Universal Robots PolyScope program: 958_16_OCT_2021_DER.urp

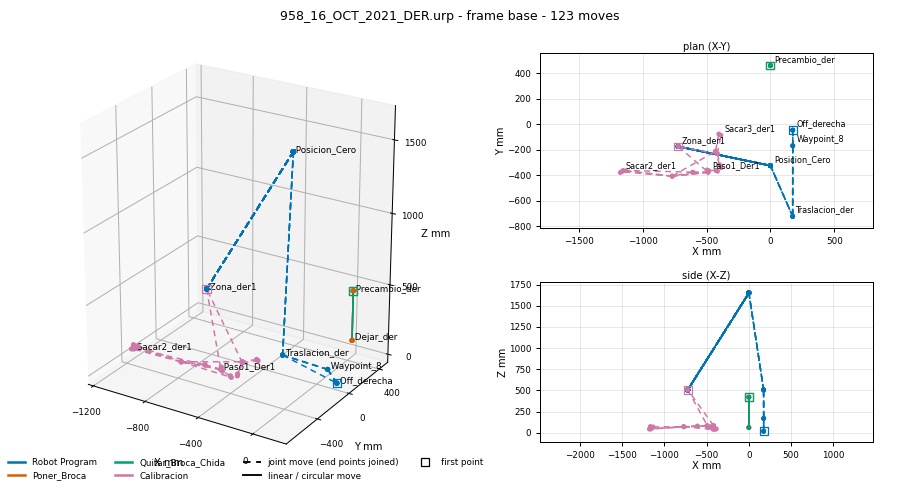
[picture p0: tool path of 958_16_OCT_2021_DER.urp in frame base, 123 of 219 moves have a stored position in this frame; points joined in program order, loops and branches not executed]
Program 958_16_OCT_2021_DER (installation=instalacion_derecha_10_MAR_21 directory=/programs/FAI3 createdIn=5.6.0.90886 lastSavedIn=5.11.1.108318 robotSerialNumber=20195001785)
Calibrated DH parameters: a=[0.000107, -0.568984, -0.552934, -0.00001, -0.000063, 0]; d=[0.180718, -257.998067, 200.685024, 57.48776, 0.119923, 0.115353]; alpha=[1.571119, 0.000876, -0.002498, 1.571178, -1.570523, 0]; deltaTheta=[0, -0.378191, 0.631587, -0.253396, 0, 0]
Robot Program (runOnlyOnce=false)
  SuppressedNode
    Folder Pruebas_Cambiador
      MoveJ speed 30 deg/s, acceleration 50 deg/s^2 (useActiveTCP=true) feature=Base
        Waypoint Precambio_der: TCP in base x=0.184 y=459.545 z=420.003 mm, rx=0.2788 ry=3.1256 rz=-0.0305 rad; joints [126.473, -59.389, -120.459, -180.773, -48.503, 0.207] deg; TCP offset x=0.151 y=-167.165 z=35.088 mm, rx=1.5784 ry=-0.0729 rz=0.0687 rad
      Loop Forever
        Call Poner_Broca
        Call Quitar_Broca_Chida
  SuppressedNode
    'Codigo'
  Set DigitalOutput pin=digital_out[0]; digitalValue=1
  MoveJ speed 30 deg/s, acceleration 50 deg/s^2 (useActiveTCP=true) feature=Base
    Waypoint Off_derecha: TCP in base x=175.178 y=-46.666 z=17.814 mm, rx=-1.9982 ry=0.0913 rz=0.0579 rad; joints [90, -90, 154.891, 0, 90, 0.001] deg
  broca := 1645
  Script: textmsg("----------DAS-----------")
  If Lado_Correr≟2
    If pos_sig_der≟0
      Folder Arranque
        Set ExpressionOutput pin=mensaje_mw10; expression=15
        Wait DigitalInput pin=Continuar_M30; digitalValue=1
        Wait Sleep waitTime=1
        MoveJ speed 60 deg/s, acceleration 80 deg/s^2 (useActiveTCP=true) feature=Base
          Waypoint Off_derecha: TCP in base x=175.178 y=-46.666 z=17.814 mm, rx=-1.9982 ry=0.0913 rz=0.0579 rad; joints [90, -90, 154.891, 0, 90, 0.001] deg
        Set DigitalOutput pin=postrnas_m187; digitalValue=1
        Wait Sleep waitTime=1
        Set DigitalOutput pin=Home_M20; digitalValue=1
        Wait Sleep waitTime=1
        Set DigitalOutput pin=postrnas_m187; digitalValue=0
        Set DigitalOutput pin=Home_M20; digitalValue=0
        Set ExpressionOutput pin=mensaje_mw10; expression=20
        Wait DigitalInput pin=Continuar_M30; digitalValue=1
        Wait Sleep waitTime=1
      Folder Traslacion
        Set ExpressionOutput pin=mensaje_mw10; expression=25
        Wait DigitalInput pin=Continuar_M30; digitalValue=1
        Wait Sleep waitTime=1
        MoveJ speed 60 deg/s, acceleration 80 deg/s^2 (useActiveTCP=true) feature=Base
          Waypoint Waypoint_8: TCP in base x=175.237 y=-168.919 z=168.903 mm, rx=3.0585 ry=-0.1387 rz=0.0062 rad; joints [90.001, -160.001, 154.893, -0.003, 90, 0.003] deg
          Waypoint Traslacion_der: TCP in base x=174.612 y=-721.747 z=506.267 mm, rx=3.1383 ry=-0.1432 rz=0.0001 rad; joints [89.991, -90.247, 90.386, -0.667, 89.974, 0.014] deg
        Set ExpressionOutput pin=mensaje_mw10; expression=30
        Wait DigitalInput pin=Continuar_M30; digitalValue=1
        Wait Sleep waitTime=1
        Set DigitalOutput pin=postrnas_m187; digitalValue=1
        Wait Sleep waitTime=1
        Set DigitalOutput pin=pose2_m252; digitalValue=1
        Wait Sleep waitTime=1
        Set DigitalOutput pin=pose2_m252; digitalValue=0
        Set DigitalOutput pin=postrnas_m187; digitalValue=0
        Wait Sleep waitTime=10
        Set ExpressionOutput pin=mensaje_mw10; expression=35
        Wait DigitalInput pin=Continuar_M30; digitalValue=1
        Wait Sleep waitTime=1
      Folder Brocas
        Set DigitalOutput pin=carrusel_home; digitalValue=1
        Wait Sleep waitTime=1
        Set DigitalOutput pin=carrusel_home; digitalValue=0
        Set ExpressionOutput pin=mensaje_mw10; expression=40
        Wait DigitalInput pin=Continuar_M30; digitalValue=1
        Wait Sleep waitTime=1
        Set DigitalOutput pin=carrusel_home; digitalValue=1
        Wait Sleep waitTime=1
        Set DigitalOutput pin=carrusel_home; digitalValue=0
        Set ExpressionOutput pin=mensaje_mw10; expression=45
        Wait DigitalInput pin=Continuar_M30; digitalValue=1
        Wait Sleep waitTime=1
        Call Poner_Broca
      Folder Offsets factor
        SuppressedNode
          broca := 1645
        L1B1x := ((0.09525254)/(0.09525))*(0.09525254)
        L1B1y := ((-0.01266698)/(-0.0127))*(-0.01266698)
        L1B2x := ((0.75576176)/(0.75565))*(0.75576176)
        L1B2y := ((-0.01269238)/(-0.0127))*(-0.01269238)
        L2B1x := ((0.09513062)/(0.09525))*(0.09525)
        L2B1y := ((0.39369238)/(0.3937))*(0.39369238)
        L2B2x := ((0.75565508)/(0.75565))*(0.75565508)
        L2B2y := ((0.39372032)/(0.3937))*(0.39372032)
      Folder Calibracion
        Set ExpressionOutput pin=mensaje_mw10; expression=50
        Wait DigitalInput pin=Continuar_M30; digitalValue=1
        Wait Sleep waitTime=1
        MoveJ speed 60 deg/s, acceleration 80 deg/s^2 (useActiveTCP=true) feature=Base
          Waypoint Posicion_Cero: TCP in base x=0.641 y=-324.742 z=1651.532 mm, rx=-0.0042 ry=-0.0154 rz=-3.0499 rad; joints [-0.001, -90.003, -0.001, -90, 0, 0.002] deg
          Waypoint Zona_der1: TCP in base x=-721.714 y=-174.597 z=506.289 mm, rx=2.1128 ry=-2.325 rz=0 rad; joints [0.057, -90.231, 90.368, -0.664, 90.292, 0.009] deg
        broca := 1645
        Set ExpressionOutput pin=mensaje_mw10; expression=125
        Wait DigitalInput pin=Continuar_M30; digitalValue=1
        Wait Sleep waitTime=1
        Set ExpressionOutput pin=mensaje_mw10; expression=130
        Wait DigitalInput pin=Continuar_M30; digitalValue=1
        Wait Sleep waitTime=1
        Call Calibracion
      Folder GoNoGo
        Set ExpressionOutput pin=mensaje_mw10; expression=55
        Wait DigitalInput pin=Continuar_M30; digitalValue=1
        Wait Sleep waitTime=1
        Set ExpressionOutput pin=mensaje_mw10; expression=60
        Wait DigitalInput pin=Continuar_M30; digitalValue=1
        Wait Sleep waitTime=1
        Folder Linea1_Buje1
          Xfin := (((L1B1x)*Xp)-(Xd)-((L1B1y)*(1/m2)))*(-1)
          Yfin := (((L1B1y)*Yp)-(Yd)+((L1B1x)*m1))*(-1)
          rotaciones := get_actual_tcp_pose()
          var_3 := rotaciones[3]
          var_4 := rotaciones[4]
          var_5 := rotaciones[5]
          If broca≟1645
            PosFinal := p[Xfin+0.00208915,Yfin+0.00208915,0.1,var_3,var_4,var_5]
          ElseIf broca≟1935
            PosFinal := p[Xfin+0.00245745,Yfin+0.00245745,0.1,var_3,var_4,var_5]
          ElseIf broca≟217
            PosFinal := p[Xfin+0.0027559,Yfin+0.0027559,0.1,var_3,var_4,var_5]
          Buje_Final := PosFinal
        MoveJ speed 60 deg/s, acceleration 80 deg/s^2 (useActiveTCP=true) feature=Base
          Waypoint Waypoint (Variable): variable(name=Buje_Final)
        Wait Sleep waitTime=1
        Folder Alturas
          If P1h[2]<P2h[2]
            tcp := get_actual_tcp_pose()
            offset_altura := p[tcp[0],tcp[1],((alta-0.0095)-(altura/1000)),tcp[3],tcp[4],tcp[5]]
            MoveL speed 250 mm/s, acceleration 1200 mm/s^2 (useActiveTCP=true) feature=Base
              Waypoint Waypoint (Variable): motionParameters(jointSpeed=1.047198 jointAcceleration=1.396263 cartesianSpeed=0.03 cartesianAcceleration=0.04); variable=offset_altura
          Else 
            tcp := get_actual_tcp_pose()
            offset_altura := p[tcp[0],tcp[1],((alta-0.0095)),tcp[3],tcp[4],tcp[5]]
            MoveL speed 250 mm/s, acceleration 1200 mm/s^2 (useActiveTCP=true) feature=Base
              Waypoint Waypoint (Variable): motionParameters(jointSpeed=1.047198 jointAcceleration=1.396263 cartesianSpeed=0.03 cartesianAcceleration=0.04); variable=offset_altura
        MoveL speed 60 mm/s, acceleration 80 mm/s^2 (useActiveTCP=true) feature=Base
          Folder Freemove
            Wait Sleep waitTime=2
            Script: freedrive_mode()
            Wait Sleep waitTime=2.5
            Script: end_freedrive_mode()
            var_11 := get_actual_tcp_pose()
            var_11 := p[var_11[0]*1000,var_11[1]*1000,420,420,420,420]
            var_11 := get_actual_tcp_pose()
            var_11 := p[var_11[0],var_11[1],0.1,var_11[3],var_11[4],var_11[5]]
          MoveDirectionNode (selectedDirection=ZPlus)
            Until DISTANCE (allowActions=false deceleration=3 distanceNodeType=STOP) Distance=0.15; motionParameters(blendRadius=0)
          MoveDirectionNode (selectedDirection=XMinus)
            Until DISTANCE (allowActions=false deceleration=3 distanceNodeType=STOP) Distance=0.42; motionParameters(blendRadius=0)
        L1B1 := var_11
        Folder Linea1_Buje2
          Xfin := (((L1B2x)*Xp)-(Xd)-((L1B2y)*(1/m2)))*(-1)
          Yfin := (((L1B2y)*Yp)-(Yd)+((L1B2x)*m1))*(-1)
          rotaciones := get_actual_tcp_pose()
          var_3 := rotaciones[3]
          var_4 := rotaciones[4]
          var_5 := rotaciones[5]
          If broca≟1645
            PosFinal := p[Xfin+0.00208915,Yfin+0.00208915,0.1,var_3,var_4,var_5]
          ElseIf broca≟1935
            PosFinal := p[Xfin+0.00245745,Yfin+0.00245745,0.1,var_3,var_4,var_5]
          ElseIf broca≟217
            PosFinal := p[Xfin+0.0027559,Yfin+0.0027559,0.1,var_3,var_4,var_5]
          Buje_Final := PosFinal
        MoveJ speed 60 deg/s, acceleration 80 deg/s^2 (useActiveTCP=true) feature=Base
          Waypoint Waypoint (Variable): variable=Buje_Final
        Wait Sleep waitTime=1
        Folder Alturas
          If P1h[2]<P2h[2]
            tcp := get_actual_tcp_pose()
            offset_altura := p[tcp[0],tcp[1],((alta-0.0095)),tcp[3],tcp[4],tcp[5]]
            MoveL speed 250 mm/s, acceleration 1200 mm/s^2 (useActiveTCP=true) feature=Base
              Waypoint Waypoint (Variable): motionParameters(jointSpeed=1.047198 jointAcceleration=1.396263 cartesianSpeed=0.03 cartesianAcceleration=0.04); variable=offset_altura
          Else 
            tcp := get_actual_tcp_pose()
            offset_altura := p[tcp[0],tcp[1],((alta-0.0095)-(altura/1000)),tcp[3],tcp[4],tcp[5]]
            MoveL speed 250 mm/s, acceleration 1200 mm/s^2 (useActiveTCP=true) feature=Base
              Waypoint Waypoint (Variable): motionParameters(jointSpeed=1.047198 jointAcceleration=1.396263 cartesianSpeed=0.03 cartesianAcceleration=0.04); variable=offset_altura
        MoveL speed 60 mm/s, acceleration 80 mm/s^2 (useActiveTCP=true) feature=Base
          Folder Freemove
            Wait Sleep waitTime=2
            Script: freedrive_mode()
            Wait Sleep waitTime=2.5
            Script: end_freedrive_mode()
            var_11 := get_actual_tcp_pose()
            var_11 := p[var_11[0]*1000,var_11[1]*1000,420,420,420,420]
            var_11 := get_actual_tcp_pose()
            var_11 := p[var_11[0],var_11[1],0.1,var_11[3],var_11[4],var_11[5]]
          MoveDirectionNode (selectedDirection=ZPlus)
            Until DISTANCE (allowActions=false deceleration=3 distanceNodeType=STOP) Distance=0.15; motionParameters(blendRadius=0)
        L1B2 := var_11
        Folder Linea2_Buje2
          Xfin := (((L2B2x)*Xp)-(Xd)-((L2B2y)*(1/m2)))*(-1)
          Yfin := (((L2B2y)*Yp)-(Yd)+((L2B2x)*m1))*(-1)
          rotaciones := get_actual_tcp_pose()
          var_3 := rotaciones[3]
          var_4 := rotaciones[4]
          var_5 := rotaciones[5]
          If broca≟1645
            PosFinal := p[Xfin+0.00208915,Yfin+0.00208915,0.1,var_3,var_4,var_5]
          ElseIf broca≟1935
            PosFinal := p[Xfin+0.00245745,Yfin+0.00245745,0.1,var_3,var_4,var_5]
          ElseIf broca≟217
            PosFinal := p[Xfin+0.0027559,Yfin+0.0027559,0.1,var_3,var_4,var_5]
          Buje_Final := PosFinal
        MoveJ speed 60 deg/s, acceleration 80 deg/s^2 (useActiveTCP=true) feature=Base
          Waypoint Waypoint (Variable): variable=Buje_Final
        Wait Sleep waitTime=1
        Folder Alturas
          If P1h[2]<P2h[2]
            tcp := get_actual_tcp_pose()
            offset_altura := p[tcp[0],tcp[1],((alta-0.0095)),tcp[3],tcp[4],tcp[5]]
            MoveL speed 250 mm/s, acceleration 1200 mm/s^2 (useActiveTCP=true) feature=Base
              Waypoint Waypoint (Variable): motionParameters(jointSpeed=1.047198 jointAcceleration=1.396263 cartesianSpeed=0.03 cartesianAcceleration=0.04); variable=offset_altura
          Else 
            tcp := get_actual_tcp_pose()
            offset_altura := p[tcp[0],tcp[1],((alta-0.0095)-(altura/1000)),tcp[3],tcp[4],tcp[5]]
            MoveL speed 250 mm/s, acceleration 1200 mm/s^2 (useActiveTCP=true) feature=Base
              Waypoint Waypoint (Variable): motionParameters(jointSpeed=1.047198 jointAcceleration=1.396263 cartesianSpeed=0.03 cartesianAcceleration=0.04); variable=offset_altura
        MoveL speed 60 mm/s, acceleration 80 mm/s^2 (useActiveTCP=true) feature=Base
          Folder Freemove
            Wait Sleep waitTime=2
            Script: freedrive_mode()
            Wait Sleep waitTime=2.5
            Script: end_freedrive_mode()
            var_11 := get_actual_tcp_pose()
            var_11 := p[var_11[0]*1000,var_11[1]*1000,420,420,420,420]
            var_11 := get_actual_tcp_pose()
            var_11 := p[var_11[0],var_11[1],0.1,var_11[3],var_11[4],var_11[5]]
          MoveDirectionNode (selectedDirection=ZPlus)
            Until DISTANCE (allowActions=false deceleration=3 distanceNodeType=STOP) Distance=0.15; motionParameters(blendRadius=0)
        L2B2 := var_11
        Folder Linea2_Buje1
          Xfin := (((L2B1x)*Xp)-(Xd)-((L2B1y)*(1/m2)))*(-1)
          Yfin := (((L2B1y)*Yp)-(Yd)+((L2B1x)*m1))*(-1)
          rotaciones := get_actual_tcp_pose()
          var_3 := rotaciones[3]
          var_4 := rotaciones[4]
          var_5 := rotaciones[5]
          If broca≟1645
            PosFinal := p[Xfin+0.00208915,Yfin+0.00208915,0.1,var_3,var_4,var_5]
          ElseIf broca≟1935
            PosFinal := p[Xfin+0.00245745,Yfin+0.00245745,0.1,var_3,var_4,var_5]
          ElseIf broca≟217
            PosFinal := p[Xfin+0.0027559,Yfin+0.0027559,0.1,var_3,var_4,var_5]
          Buje_Final := PosFinal
        MoveJ speed 60 deg/s, acceleration 80 deg/s^2 (useActiveTCP=true) feature=Base
          Waypoint Waypoint (Variable): variable=Buje_Final
        Wait Sleep waitTime=1
        Folder Alturas
          If P1h[2]<P2h[2]
            tcp := get_actual_tcp_pose()
            offset_altura := p[tcp[0],tcp[1],((alta-0.0095)-(altura/1000)),tcp[3],tcp[4],tcp[5]]
            MoveL speed 250 mm/s, acceleration 1200 mm/s^2 (useActiveTCP=true) feature=Base
              Waypoint Waypoint (Variable): motionParameters(jointSpeed=1.047198 jointAcceleration=1.396263 cartesianSpeed=0.03 cartesianAcceleration=0.04); variable=offset_altura
          Else 
            tcp := get_actual_tcp_pose()
            offset_altura := p[tcp[0],tcp[1],((alta-0.0095)),tcp[3],tcp[4],tcp[5]]
            MoveL speed 250 mm/s, acceleration 1200 mm/s^2 (useActiveTCP=true) feature=Base
              Waypoint Waypoint (Variable): motionParameters(jointSpeed=1.047198 jointAcceleration=1.396263 cartesianSpeed=0.03 cartesianAcceleration=0.04); variable=offset_altura
        MoveL speed 60 mm/s, acceleration 80 mm/s^2 (useActiveTCP=true) feature=Base
          Folder Freemove
            Wait Sleep waitTime=2
            Script: freedrive_mode()
            Wait Sleep waitTime=2.5
            Script: end_freedrive_mode()
            var_11 := get_actual_tcp_pose()
            var_11 := p[var_11[0]*1000,var_11[1]*1000,420,420,420,420]
            var_11 := get_actual_tcp_pose()
            var_11 := p[var_11[0],var_11[1],0.1,var_11[3],var_11[4],var_11[5]]
          MoveDirectionNode (selectedDirection=ZPlus)
            Until DISTANCE (allowActions=false deceleration=3 distanceNodeType=STOP) Distance=0.15; motionParameters(blendRadius=0)
        L2B1 := var_11
        MoveJ speed 60 deg/s, acceleration 80 deg/s^2 (useActiveTCP=true) feature=Base
          Waypoint Zona_der1: TCP in base x=-721.714 y=-174.597 z=506.289 mm, rx=2.1128 ry=-2.325 rz=0 rad; joints [0.057, -90.231, 90.368, -0.664, 90.292, 0.009] deg
      Folder Colocar broca
        Call Quitar_Broca_Chida
        Call Poner_Broca
      SuppressedNode
        Folder Cancelar barrenacion
          MoveJ speed 60 deg/s, acceleration 80 deg/s^2 (useActiveTCP=true) feature=Base
            Waypoint Zona_der1: TCP in base x=-721.714 y=-174.597 z=506.289 mm, rx=2.1128 ry=-2.325 rz=0 rad; joints [0.057, -90.231, 90.368, -0.664, 90.292, 0.009] deg
            Waypoint Posicion_Cero: TCP in base x=0.641 y=-324.742 z=1651.532 mm, rx=-0.0042 ry=-0.0154 rz=-3.0499 rad; joints [-0.001, -90.003, -0.001, -90, 0, 0.002] deg
          Call Quitar_Broca_Chida
          Set DigitalOutput pin=lado_hecho; digitalValue=1
          Set ExpressionOutput pin=mensaje_mw10; expression=100
          Wait DigitalInput pin=Continuar_M30; digitalValue=1
          Wait Sleep waitTime=1
          Set ExpressionOutput pin=mensaje_mw10; expression=155
          Wait DigitalInput pin=Continuar_M30; digitalValue=1
          Wait Sleep waitTime=1
          Set ExpressionOutput pin=mensaje_mw10; expression=35
          Wait DigitalInput pin=Continuar_M30; digitalValue=1
          Wait Sleep waitTime=1
      Folder Barrenado
        Set ExpressionOutput pin=mensaje_mw10; expression=65
        Wait DigitalInput pin=Continuar_M30; digitalValue=1
        Wait Sleep waitTime=1
        Set ExpressionOutput pin=mensaje_mw10; expression=150
        Wait Sleep waitTime=1
        Folder Linea 1 a 1645
          broca := 1645
          Folder Buje_inicial
            Buje_Inicial := L1B2
          Folder Buje_final
            Buje_Final := L1B1
          barrenosTotales := 27
          barrenoActual := 1
          Loop While (checkContinuously=false) expression=barrenoActual≤barrenosTotales
            MoveL speed 250 mm/s, acceleration 1200 mm/s^2 (useActiveTCP=true) feature=Base
              bajada_broca := p[0,0,0.006,0,0,0]
              internos := interpolate_pose(Buje_Inicial, Buje_Final, ((barrenoActual)-1)/((barrenosTotales)-1))
              If barrenoActual≟1 or barrenoActual≟3 or barrenoActual≟5 or barrenoActual≟7 or barrenoActual≟9 or barrenoActual≟11 or barrenoActual≟13 or barrenoActual≟15 or barrenoActual≟17 or barrenoActual≟19 or barrenoActual≟21 or barrenoActual≟23 or barrenoActual≟25 or barrenoActual≟27
                Set ExpressionOutput pin=mensaje_mw10; expression=200
                Wait DigitalInput pin=Continuar_M30; digitalValue=1
                Wait Sleep waitTime=1
                Set ExpressionOutput pin=mensaje_mw10; expression=150
                Wait Sleep waitTime=1
              MoveJ speed 30 deg/s, acceleration 40 deg/s^2 (useActiveTCP=true) feature=Base
                Waypoint Waypoint (Variable): variable(name=internos)
              Wait Sleep waitTime=2
              Folder Alturas
                If P1h[2]<P2h[2]
                  acomodo := (altura/(barrenosTotales-1))*(barrenoActual-1)
                  tcp := get_actual_tcp_pose()
                  offset_altura := p[tcp[0],tcp[1],((alta-0.0095)-(acomodo/1000)),tcp[3],tcp[4],tcp[5]]
                  MoveL speed 250 mm/s, acceleration 1200 mm/s^2 (useActiveTCP=true) feature=Base
                    Waypoint Waypoint (Variable): motionParameters(jointSpeed=1.047198 jointAcceleration=1.396263 cartesianSpeed=0.03 cartesianAcceleration=0.04); variable=offset_altura
                Else 
                  acomodo := (altura/(barrenosTotales-1))*(26-(barrenoActual-1))
                  tcp := get_actual_tcp_pose()
                  offset_altura := p[tcp[0],tcp[1],((alta-0.0095)-(acomodo/1000)),tcp[3],tcp[4],tcp[5]]
                  MoveL speed 250 mm/s, acceleration 1200 mm/s^2 (useActiveTCP=true) feature=Base
                    Waypoint Waypoint (Variable): motionParameters(jointSpeed=1.047198 jointAcceleration=1.396263 cartesianSpeed=0.03 cartesianAcceleration=0.04); variable=offset_altura
              Folder Freemove
                Wait Sleep waitTime=2
                Script: freedrive_mode()
                Wait Sleep waitTime=2.5
                Script: end_freedrive_mode()
              Wait Sleep waitTime=0.3
              Set DigitalOutput pin=config_out[1]; digitalValue=1
              Wait Sleep waitTime=1
              Wait Sleep waitTime=0.3
              Wait Sleep waitTime=0.3
              Wait Sleep waitTime=0.3
              Loop Counting (count=3) loopVariable(name=Loop_59)
                Poses_taladrado := pose_sub(get_actual_tcp_pose(), bajada_broca)
                Waypoint Waypoint (Variable): motionParameters(jointSpeed=1.047198 jointAcceleration=1.396263 cartesianSpeed=0.001 cartesianAcceleration=0.005); variable(name=Poses_taladrado)
                If bajada_broca≟p[0,0,0.018,0,0,0]
                  num_barreno := str_cat("Barreno: ",barrenoActual)
                  tcp_actual := get_actual_tcp_pose()
                  X_actual := str_cat("     X: ",tcp_actual[0])
                  Y_actual := str_cat("     Y: ",tcp_actual[1])
                  pos_barreno := str_cat(X_actual,Y_actual)
                  Script: textmsg(num_barreno,pos_barreno)
                Poses_taladrado := pose_add(get_actual_tcp_pose(), bajada_broca)
                Waypoint Waypoint (Variable): motionParameters(jointSpeed=1.047198 jointAcceleration=1.396263 cartesianSpeed=0.01 cartesianAcceleration=0.01); variable=Poses_taladrado
                bajada_broca := pose_add(bajada_broca, p[0,0,0.006,0,0,0])
              MoveDirectionNode (selectedDirection=ZPlus toolParams=0.03, 0.04)
                Until DISTANCE (allowActions=false deceleration=3 distanceNodeType=STOP) Distance=0.05; motionParameters(blendRadius=0)
              MoveJ speed 30 deg/s, acceleration 40 deg/s^2 (useActiveTCP=true) feature=Base
                Waypoint Waypoint (Variable): variable=internos
              Wait Sleep waitTime=0.3
              Set DigitalOutput pin=config_out[1]; digitalValue=0
              Wait Sleep waitTime=0.3
              If barrenoActual≟13 or barrenoActual≟27
                MoveDirectionNode (selectedDirection=ZPlus toolParams=0.03, 0.04)
                  Until DISTANCE (allowActions=false deceleration=3 distanceNodeType=STOP) Distance=0.03; motionParameters(blendRadius=0)
                MoveJ speed 30 deg/s, acceleration 40 deg/s^2 (useActiveTCP=true) feature=Base
                  Waypoint Zona_der1: TCP in base x=-721.714 y=-174.597 z=506.289 mm, rx=2.1128 ry=-2.325 rz=0 rad; joints [0.057, -90.231, 90.368, -0.664, 90.292, 0.009] deg
                  Waypoint Posicion_Cero: TCP in base x=0.641 y=-324.742 z=1651.532 mm, rx=-0.0042 ry=-0.0154 rz=-3.0499 rad; joints [-0.001, -90.003, -0.001, -90, 0, 0.002] deg
                Call Quitar_Broca_Chida
                If barrenoActual≟13
                  Call Poner_Broca
                ElseIf barrenoActual≟27
                  Call Poner_Broca
                MoveJ speed 30 deg/s, acceleration 40 deg/s^2 (useActiveTCP=true) feature=Base
                  Waypoint Posicion_Cero: TCP in base x=0.641 y=-324.742 z=1651.532 mm, rx=-0.0042 ry=-0.0154 rz=-3.0499 rad; joints [-0.001, -90.003, -0.001, -90, 0, 0.002] deg
                  Waypoint Zona_der1: TCP in base x=-721.714 y=-174.597 z=506.289 mm, rx=2.1128 ry=-2.325 rz=0 rad; joints [0.057, -90.231, 90.368, -0.664, 90.292, 0.009] deg
              barrenoActual := barrenoActual+1
        Folder Linea 2 a 1645
          broca := 1645
          Folder Buje_inicial
            Buje_Inicial := L2B2
          Folder Buje_final
            Buje_Final := L2B1
          barrenosTotales := 27
          barrenoActual := 1
          Loop While (checkContinuously=false) expression=barrenoActual≤barrenosTotales
            MoveL speed 250 mm/s, acceleration 1200 mm/s^2 (useActiveTCP=true) feature=Base
              bajada_broca := p[0,0,0.006,0,0,0]
              internos := interpolate_pose(Buje_Inicial, Buje_Final, ((barrenoActual)-1)/((barrenosTotales)-1))
              Folder Alturas
                If barrenoActual≟1 or barrenoActual≟3 or barrenoActual≟5 or barrenoActual≟7 or barrenoActual≟9 or barrenoActual≟11 or barrenoActual≟13 or barrenoActual≟15 or barrenoActual≟17 or barrenoActual≟19 or barrenoActual≟21 or barrenoActual≟23 or barrenoActual≟25 or barrenoActual≟27
                  Set ExpressionOutput pin=mensaje_mw10; expression=200
                  Wait DigitalInput pin=Continuar_M30; digitalValue=1
                  Wait Sleep waitTime=1
                  Set ExpressionOutput pin=mensaje_mw10; expression=150
                  Wait Sleep waitTime=1
                MoveJ speed 30 deg/s, acceleration 40 deg/s^2 (useActiveTCP=true) feature=Base
                  Waypoint Waypoint (Variable): variable=internos
                Wait Sleep waitTime=2
                If P1h[2]<P2h[2]
                  acomodo := (altura/(barrenosTotales-1))*(barrenoActual-1)
                  tcp := get_actual_tcp_pose()
                  offset_altura := p[tcp[0],tcp[1],((alta-0.0095)-(acomodo/1000)),tcp[3],tcp[4],tcp[5]]
                  MoveL speed 250 mm/s, acceleration 1200 mm/s^2 (useActiveTCP=true) feature=Base
                    Waypoint Waypoint (Variable): motionParameters(jointSpeed=1.047198 jointAcceleration=1.396263 cartesianSpeed=0.03 cartesianAcceleration=0.04); variable=offset_altura
                Else 
                  acomodo := (altura/(barrenosTotales-1))*(26-(barrenoActual-1))
                  tcp := get_actual_tcp_pose()
                  offset_altura := p[tcp[0],tcp[1],((alta-0.0095)-(acomodo/1000)),tcp[3],tcp[4],tcp[5]]
                  MoveL speed 250 mm/s, acceleration 1200 mm/s^2 (useActiveTCP=true) feature=Base
                    Waypoint Waypoint (Variable): motionParameters(jointSpeed=1.047198 jointAcceleration=1.396263 cartesianSpeed=0.03 cartesianAcceleration=0.04); variable=offset_altura
              Folder Freemove
                Wait Sleep waitTime=2
                Script: freedrive_mode()
                Wait Sleep waitTime=2.5
                Script: end_freedrive_mode()
              Wait Sleep waitTime=0.3
              Set DigitalOutput pin=config_out[1]; digitalValue=1
              Wait Sleep waitTime=1
              Wait Sleep waitTime=0.3
              Wait Sleep waitTime=0.3
              Wait Sleep waitTime=0.3
              Loop Counting (count=3) loopVariable(name=Loop_61)
                Poses_taladrado := pose_sub(get_actual_tcp_pose(), bajada_broca)
                Waypoint Waypoint (Variable): motionParameters(jointSpeed=1.047198 jointAcceleration=1.396263 cartesianSpeed=0.001 cartesianAcceleration=0.005); variable=Poses_taladrado
                If bajada_broca≟p[0,0,0.018,0,0,0]
                  num_barreno := str_cat("Barreno: ",barrenoActual)
                  tcp_actual := get_actual_tcp_pose()
                  X_actual := str_cat("     X: ",tcp_actual[0])
                  Y_actual := str_cat("     Y: ",tcp_actual[1])
                  pos_barreno := str_cat(X_actual,Y_actual)
                  Script: textmsg(num_barreno,pos_barreno)
                Poses_taladrado := pose_add(get_actual_tcp_pose(), bajada_broca)
                Waypoint Waypoint (Variable): motionParameters(jointSpeed=1.047198 jointAcceleration=1.396263 cartesianSpeed=0.01 cartesianAcceleration=0.01); variable=Poses_taladrado
                bajada_broca := pose_add(bajada_broca, p[0,0,0.006,0,0,0])
              MoveDirectionNode (selectedDirection=ZPlus toolParams=0.03, 0.04)
                Until DISTANCE (allowActions=false deceleration=3 distanceNodeType=STOP) Distance=0.05; motionParameters(blendRadius=0)
              MoveJ speed 30 deg/s, acceleration 40 deg/s^2 (useActiveTCP=true) feature=Base
                Waypoint Waypoint (Variable): variable=internos
              Wait Sleep waitTime=0.3
              Set DigitalOutput pin=config_out[1]; digitalValue=0
              Wait Sleep waitTime=0.3
              If barrenoActual≟13
                MoveDirectionNode (selectedDirection=ZPlus)
                  Until DISTANCE (allowActions=false deceleration=3 distanceNodeType=STOP) Distance=0.03; motionParameters(blendRadius=0)
                MoveJ speed 60 deg/s, acceleration 80 deg/s^2 (useActiveTCP=true) feature=Base
                  Waypoint Zona_der1: TCP in base x=-721.714 y=-174.597 z=506.289 mm, rx=2.1128 ry=-2.325 rz=0 rad; joints [0.057, -90.231, 90.368, -0.664, 90.292, 0.009] deg
                  Waypoint Posicion_Cero: TCP in base x=0.641 y=-324.742 z=1651.532 mm, rx=-0.0042 ry=-0.0154 rz=-3.0499 rad; joints [-0.001, -90.003, -0.001, -90, 0, 0.002] deg
                Call Quitar_Broca_Chida
                Call Poner_Broca
                MoveJ speed 60 deg/s, acceleration 80 deg/s^2 (useActiveTCP=true) feature=Base
                  Waypoint Posicion_Cero: TCP in base x=0.641 y=-324.742 z=1651.532 mm, rx=-0.0042 ry=-0.0154 rz=-3.0499 rad; joints [-0.001, -90.003, -0.001, -90, 0, 0.002] deg
                  Waypoint Zona_der1: TCP in base x=-721.714 y=-174.597 z=506.289 mm, rx=2.1128 ry=-2.325 rz=0 rad; joints [0.057, -90.231, 90.368, -0.664, 90.292, 0.009] deg
              ElseIf barrenoActual≟27
                MoveDirectionNode (selectedDirection=ZPlus)
                  Until DISTANCE (allowActions=false deceleration=3 distanceNodeType=STOP) Distance=0.03; motionParameters(blendRadius=0)
                MoveJ speed 60 deg/s, acceleration 80 deg/s^2 (useActiveTCP=true) feature=Base
                  Waypoint Zona_der1: TCP in base x=-721.714 y=-174.597 z=506.289 mm, rx=2.1128 ry=-2.325 rz=0 rad; joints [0.057, -90.231, 90.368, -0.664, 90.292, 0.009] deg
                  Waypoint Posicion_Cero: TCP in base x=0.641 y=-324.742 z=1651.532 mm, rx=-0.0042 ry=-0.0154 rz=-3.0499 rad; joints [-0.001, -90.003, -0.001, -90, 0, 0.002] deg
                Call Quitar_Broca_Chida
                Set DigitalOutput pin=carrusel_home; digitalValue=1
                Wait Sleep waitTime=1
                Set DigitalOutput pin=carrusel_home; digitalValue=0
                Set ExpressionOutput pin=mensaje_mw10; expression=70
                Wait DigitalInput pin=Continuar_M30; digitalValue=1
                Wait Sleep waitTime=1
                Set ExpressionOutput pin=mensaje_mw10; expression=120
                Wait DigitalInput pin=Continuar_M30; digitalValue=1
                Wait Sleep waitTime=1
                Set DigitalOutput pin=carrusel_home; digitalValue=1
                Wait Sleep waitTime=1
                Set DigitalOutput pin=carrusel_home; digitalValue=0
                Set ExpressionOutput pin=mensaje_mw10; expression=75
                Wait DigitalInput pin=Continuar_M30; digitalValue=1
                Wait Sleep waitTime=1
                Call Poner_Broca
                broca := 1935
                MoveJ speed 60 deg/s, acceleration 80 deg/s^2 (useActiveTCP=true) feature=Base
                  Waypoint Posicion_Cero: TCP in base x=0.641 y=-324.742 z=1651.532 mm, rx=-0.0042 ry=-0.0154 rz=-3.0499 rad; joints [-0.001, -90.003, -0.001, -90, 0, 0.002] deg
                  Waypoint Zona_der1: TCP in base x=-721.714 y=-174.597 z=506.289 mm, rx=2.1128 ry=-2.325 rz=0 rad; joints [0.057, -90.231, 90.368, -0.664, 90.292, 0.009] deg
                Set ExpressionOutput pin=mensaje_mw10; expression=80
                Wait DigitalInput pin=Continuar_M30; digitalValue=1
                Wait Sleep waitTime=1
                Set ExpressionOutput pin=mensaje_mw10; expression=150
                Wait DigitalInput pin=Continuar_M30; digitalValue=1
                Wait Sleep waitTime=1
              barrenoActual := barrenoActual+1
        Folder Linea 1 a 1935
          broca := 1935
          Folder Buje_inicial
            Buje_Inicial := L1B2
          Folder Buje_final
            Buje_Final := L1B1
          barrenosTotales := 27
          barrenoActual := 1
          Loop While (checkContinuously=false) expression=barrenoActual≤barrenosTotales
            MoveL speed 250 mm/s, acceleration 1200 mm/s^2 (useActiveTCP=true) feature=Base
              bajada_broca := p[0,0,0.009,0,0,0]
              internos := interpolate_pose(Buje_Inicial, Buje_Final, ((barrenoActual)-1)/((barrenosTotales)-1))
              Folder Alturas
                If barrenoActual≟1 or barrenoActual≟3 or barrenoActual≟5 or barrenoActual≟7 or barrenoActual≟9 or barrenoActual≟11 or barrenoActual≟13 or barrenoActual≟15 or barrenoActual≟17 or barrenoActual≟19 or barrenoActual≟21 or barrenoActual≟23 or barrenoActual≟25 or barrenoActual≟27
                  Set ExpressionOutput pin=mensaje_mw10; expression=200
                  Wait DigitalInput pin=Continuar_M30; digitalValue=1
                  Wait Sleep waitTime=1
                  Set ExpressionOutput pin=mensaje_mw10; expression=150
                  Wait Sleep waitTime=1
                MoveJ speed 30 deg/s, acceleration 40 deg/s^2 (useActiveTCP=true) feature=Base
                  Waypoint Waypoint (Variable): variable=internos
                Wait Sleep waitTime=2
                If P1h[2]<P2h[2]
                  acomodo := (altura/(barrenosTotales-1))*(barrenoActual-1)
                  tcp := get_actual_tcp_pose()
                  offset_altura := p[tcp[0],tcp[1],((alta-0.0095)-(acomodo/1000)),tcp[3],tcp[4],tcp[5]]
                  MoveL speed 250 mm/s, acceleration 1200 mm/s^2 (useActiveTCP=true) feature=Base
                    Waypoint Waypoint (Variable): motionParameters(jointSpeed=1.047198 jointAcceleration=1.396263 cartesianSpeed=0.03 cartesianAcceleration=0.04); variable=offset_altura
                Else 
                  acomodo := (altura/(barrenosTotales-1))*(26-(barrenoActual-1))
                  tcp := get_actual_tcp_pose()
                  offset_altura := p[tcp[0],tcp[1],((alta-0.0095)-(acomodo/1000)),tcp[3],tcp[4],tcp[5]]
                  MoveL speed 250 mm/s, acceleration 1200 mm/s^2 (useActiveTCP=true) feature=Base
                    Waypoint Waypoint (Variable): motionParameters(jointSpeed=1.047198 jointAcceleration=1.396263 cartesianSpeed=0.03 cartesianAcceleration=0.04); variable=offset_altura
              Folder Freemove
                Wait Sleep waitTime=2
                Script: freedrive_mode()
                Wait Sleep waitTime=2.5
                Script: end_freedrive_mode()
              Wait Sleep waitTime=0.3
              Set DigitalOutput pin=config_out[1]; digitalValue=1
              Wait Sleep waitTime=1
              Wait Sleep waitTime=0.3
              Wait Sleep waitTime=0.3
              Wait Sleep waitTime=0.3
              Loop Counting (count=2) loopVariable(name=Loop_63)
                Poses_taladrado := pose_sub(get_actual_tcp_pose(), bajada_broca)
                Waypoint Waypoint (Variable): motionParameters(jointSpeed=1.047198 jointAcceleration=1.396263 cartesianSpeed=0.001 cartesianAcceleration=0.005); variable=Poses_taladrado
                If bajada_broca≟p[0,0,0.018,0,0,0]
                  num_barreno := str_cat("Barreno: ",barrenoActual)
                  tcp_actual := get_actual_tcp_pose()
                  X_actual := str_cat("     X: ",tcp_actual[0])
                  Y_actual := str_cat("     Y: ",tcp_actual[1])
                  pos_barreno := str_cat(X_actual,Y_actual)
                  Script: textmsg(num_barreno,pos_barreno)
                Poses_taladrado := pose_add(get_actual_tcp_pose(), bajada_broca)
                Waypoint Waypoint (Variable): motionParameters(jointSpeed=1.047198 jointAcceleration=1.396263 cartesianSpeed=0.01 cartesianAcceleration=0.01); variable=Poses_taladrado
                bajada_broca := pose_add(bajada_broca, p[0,0,0.009,0,0,0])
              MoveDirectionNode (selectedDirection=ZPlus toolParams=0.01, 0.01)
                Until DISTANCE (allowActions=false deceleration=3 distanceNodeType=STOP) Distance=0.05; motionParameters(blendRadius=0)
              MoveJ speed 30 deg/s, acceleration 40 deg/s^2 (useActiveTCP=true) feature=Base
                Waypoint Waypoint (Variable): variable=internos
              Wait Sleep waitTime=0.3
              Set DigitalOutput pin=config_out[1]; digitalValue=0
              Wait Sleep waitTime=0.3
              If barrenoActual≟13 or barrenoActual≟27
                MoveDirectionNode (selectedDirection=ZPlus toolParams=0.03, 0.04)
                  Until DISTANCE (allowActions=false deceleration=3 distanceNodeType=STOP) Distance=0.03; motionParameters(blendRadius=0)
                MoveJ speed 30 deg/s, acceleration 40 deg/s^2 (useActiveTCP=true) feature=Base
                  Waypoint Zona_der1: TCP in base x=-721.714 y=-174.597 z=506.289 mm, rx=2.1128 ry=-2.325 rz=0 rad; joints [0.057, -90.231, 90.368, -0.664, 90.292, 0.009] deg
                  Waypoint Posicion_Cero: TCP in base x=0.641 y=-324.742 z=1651.532 mm, rx=-0.0042 ry=-0.0154 rz=-3.0499 rad; joints [-0.001, -90.003, -0.001, -90, 0, 0.002] deg
                Call Quitar_Broca_Chida
                If barrenoActual≟13
                  Call Poner_Broca
                ElseIf barrenoActual≟27
                  Call Poner_Broca
                MoveJ speed 30 deg/s, acceleration 40 deg/s^2 (useActiveTCP=true) feature=Base
                  Waypoint Posicion_Cero: TCP in base x=0.641 y=-324.742 z=1651.532 mm, rx=-0.0042 ry=-0.0154 rz=-3.0499 rad; joints [-0.001, -90.003, -0.001, -90, 0, 0.002] deg
                  Waypoint Zona_der1: TCP in base x=-721.714 y=-174.597 z=506.289 mm, rx=2.1128 ry=-2.325 rz=0 rad; joints [0.057, -90.231, 90.368, -0.664, 90.292, 0.009] deg
              barrenoActual := barrenoActual+1
        Folder Linea 2 a 1935
          broca := 1935
          Folder Buje_inicial
            Buje_Inicial := L2B2
          Folder Buje_final
            Buje_Final := L2B1
          barrenosTotales := 27
          barrenoActual := 1
          Loop While (checkContinuously=false) expression=barrenoActual≤barrenosTotales
            MoveL speed 250 mm/s, acceleration 1200 mm/s^2 (useActiveTCP=true) feature=Base
              bajada_broca := p[0,0,0.009,0,0,0]
              internos := interpolate_pose(Buje_Inicial, Buje_Final, ((barrenoActual)-1)/((barrenosTotales)-1))
              Folder Alturas
                If barrenoActual≟1 or barrenoActual≟3 or barrenoActual≟5 or barrenoActual≟7 or barrenoActual≟9 or barrenoActual≟11 or barrenoActual≟13 or barrenoActual≟15 or barrenoActual≟17 or barrenoActual≟19 or barrenoActual≟21 or barrenoActual≟23 or barrenoActual≟25 or barrenoActual≟27
                  Set ExpressionOutput pin=mensaje_mw10; expression=200
                  Wait DigitalInput pin=Continuar_M30; digitalValue=1
                  Wait Sleep waitTime=1
                  Set ExpressionOutput pin=mensaje_mw10; expression=150
                  Wait Sleep waitTime=1
                MoveJ speed 30 deg/s, acceleration 40 deg/s^2 (useActiveTCP=true) feature=Base
                  Waypoint Waypoint (Variable): variable=internos
                Wait Sleep waitTime=2
                If P1h[2]<P2h[2]
                  acomodo := (altura/(barrenosTotales-1))*(barrenoActual-1)
                  tcp := get_actual_tcp_pose()
                  offset_altura := p[tcp[0],tcp[1],((alta-0.0095)-(acomodo/1000)),tcp[3],tcp[4],tcp[5]]
                  MoveL speed 250 mm/s, acceleration 1200 mm/s^2 (useActiveTCP=true) feature=Base
                    Waypoint Waypoint (Variable): motionParameters(jointSpeed=1.047198 jointAcceleration=1.396263 cartesianSpeed=0.03 cartesianAcceleration=0.04); variable=offset_altura
                Else 
                  acomodo := (altura/(barrenosTotales-1))*(26-(barrenoActual-1))
                  tcp := get_actual_tcp_pose()
                  offset_altura := p[tcp[0],tcp[1],((alta-0.0095)-(acomodo/1000)),tcp[3],tcp[4],tcp[5]]
                  MoveL speed 250 mm/s, acceleration 1200 mm/s^2 (useActiveTCP=true) feature=Base
                    Waypoint Waypoint (Variable): motionParameters(jointSpeed=1.047198 jointAcceleration=1.396263 cartesianSpeed=0.03 cartesianAcceleration=0.04); variable=offset_altura
              Folder Freemove
                Wait Sleep waitTime=2
                Script: freedrive_mode()
                Wait Sleep waitTime=2.5
                Script: end_freedrive_mode()
              Wait Sleep waitTime=0.3
              Set DigitalOutput pin=config_out[1]; digitalValue=1
              Wait Sleep waitTime=1
              Wait Sleep waitTime=0.3
              Wait Sleep waitTime=0.3
              Wait Sleep waitTime=0.3
              Loop Counting (count=2) loopVariable(name=Loop_65)
                Poses_taladrado := pose_sub(get_actual_tcp_pose(), bajada_broca)
                Waypoint Waypoint (Variable): motionParameters(jointSpeed=1.047198 jointAcceleration=1.396263 cartesianSpeed=0.001 cartesianAcceleration=0.005); variable=Poses_taladrado
                If bajada_broca≟p[0,0,0.018,0,0,0]
                  num_barreno := str_cat("Barreno: ",barrenoActual)
                  tcp_actual := get_actual_tcp_pose()
                  X_actual := str_cat("     X: ",tcp_actual[0])
                  Y_actual := str_cat("     Y: ",tcp_actual[1])
                  pos_barreno := str_cat(X_actual,Y_actual)
                  Script: textmsg(num_barreno,pos_barreno)
                Poses_taladrado := pose_add(get_actual_tcp_pose(), bajada_broca)
                Waypoint Waypoint (Variable): motionParameters(jointSpeed=1.047198 jointAcceleration=1.396263 cartesianSpeed=0.01 cartesianAcceleration=0.01); variable=Poses_taladrado
                bajada_broca := pose_add(bajada_broca, p[0,0,0.009,0,0,0])
              MoveDirectionNode (selectedDirection=ZPlus toolParams=0.01, 0.01)
                Until DISTANCE (allowActions=false deceleration=3 distanceNodeType=STOP) Distance=0.05; motionParameters(blendRadius=0)
              MoveJ speed 30 deg/s, acceleration 40 deg/s^2 (useActiveTCP=true) feature=Base
                Waypoint Waypoint (Variable): variable=internos
              Wait Sleep waitTime=0.3
              Set DigitalOutput pin=config_out[1]; digitalValue=0
              Wait Sleep waitTime=0.3
              If barrenoActual≟13
                MoveDirectionNode (selectedDirection=ZPlus toolParams=0.03, 0.04)
                  Until DISTANCE (allowActions=false deceleration=3 distanceNodeType=STOP) Distance=0.03; motionParameters(blendRadius=0)
                MoveJ speed 60 deg/s, acceleration 80 deg/s^2 (useActiveTCP=true) feature=Base
                  Waypoint Zona_der1: TCP in base x=-721.714 y=-174.597 z=506.289 mm, rx=2.1128 ry=-2.325 rz=0 rad; joints [0.057, -90.231, 90.368, -0.664, 90.292, 0.009] deg
                  Waypoint Posicion_Cero: TCP in base x=0.641 y=-324.742 z=1651.532 mm, rx=-0.0042 ry=-0.0154 rz=-3.0499 rad; joints [-0.001, -90.003, -0.001, -90, 0, 0.002] deg
                Call Quitar_Broca_Chida
                Call Poner_Broca
                MoveJ speed 60 deg/s, acceleration 80 deg/s^2 (useActiveTCP=true) feature=Base
                  Waypoint Posicion_Cero: TCP in base x=0.641 y=-324.742 z=1651.532 mm, rx=-0.0042 ry=-0.0154 rz=-3.0499 rad; joints [-0.001, -90.003, -0.001, -90, 0, 0.002] deg
                  Waypoint Zona_der1: TCP in base x=-721.714 y=-174.597 z=506.289 mm, rx=2.1128 ry=-2.325 rz=0 rad; joints [0.057, -90.231, 90.368, -0.664, 90.292, 0.009] deg
              ElseIf barrenoActual≟27
                MoveDirectionNode (selectedDirection=ZPlus toolParams=0.03, 0.04)
                  Until DISTANCE (allowActions=false deceleration=3 distanceNodeType=STOP) Distance=0.03; motionParameters(blendRadius=0)
                MoveJ speed 60 deg/s, acceleration 80 deg/s^2 (useActiveTCP=true) feature=Base
                  Waypoint Zona_der1: TCP in base x=-721.714 y=-174.597 z=506.289 mm, rx=2.1128 ry=-2.325 rz=0 rad; joints [0.057, -90.231, 90.368, -0.664, 90.292, 0.009] deg
                  Waypoint Posicion_Cero: TCP in base x=0.641 y=-324.742 z=1651.532 mm, rx=-0.0042 ry=-0.0154 rz=-3.0499 rad; joints [-0.001, -90.003, -0.001, -90, 0, 0.002] deg
                Call Quitar_Broca_Chida
                Set DigitalOutput pin=carrusel_home; digitalValue=1
                Wait Sleep waitTime=1
                Set DigitalOutput pin=carrusel_home; digitalValue=0
                Set ExpressionOutput pin=mensaje_mw10; expression=85
                Wait DigitalInput pin=Continuar_M30; digitalValue=1
                Wait Sleep waitTime=1
                Set ExpressionOutput pin=mensaje_mw10; expression=120
                Wait DigitalInput pin=Continuar_M30; digitalValue=1
                Wait Sleep waitTime=1
                Set DigitalOutput pin=carrusel_home; digitalValue=1
                Wait Sleep waitTime=1
                Set DigitalOutput pin=carrusel_home; digitalValue=0
                Set ExpressionOutput pin=mensaje_mw10; expression=90
                Wait DigitalInput pin=Continuar_M30; digitalValue=1
                Wait Sleep waitTime=1
                Call Poner_Broca
                broca := 217
                MoveJ speed 60 deg/s, acceleration 80 deg/s^2 (useActiveTCP=true) feature=Base
                  Waypoint Posicion_Cero: TCP in base x=0.641 y=-324.742 z=1651.532 mm, rx=-0.0042 ry=-0.0154 rz=-3.0499 rad; joints [-0.001, -90.003, -0.001, -90, 0, 0.002] deg
                  Waypoint Zona_der1: TCP in base x=-721.714 y=-174.597 z=506.289 mm, rx=2.1128 ry=-2.325 rz=0 rad; joints [0.057, -90.231, 90.368, -0.664, 90.292, 0.009] deg
                Set ExpressionOutput pin=mensaje_mw10; expression=95
                Wait DigitalInput pin=Continuar_M30; digitalValue=1
                Wait Sleep waitTime=1
                Set ExpressionOutput pin=mensaje_mw10; expression=150
                Wait DigitalInput pin=Continuar_M30; digitalValue=1
                Wait Sleep waitTime=1
              barrenoActual := barrenoActual+1
        Folder Linea 1 a 217
          broca := 217
          Folder Buje_inicial
            Buje_Inicial := L1B2
          Folder Buje_final
            Buje_Final := L1B1
          barrenosTotales := 27
          barrenoActual := 1
          Loop While (checkContinuously=false) expression=barrenoActual≤barrenosTotales
            MoveL speed 250 mm/s, acceleration 1200 mm/s^2 (useActiveTCP=true) feature=Base
              bajada_broca := p[0,0,0.018,0,0,0]
              internos := interpolate_pose(Buje_Inicial, Buje_Final, ((barrenoActual)-1)/((barrenosTotales)-1))
              Wait Sleep waitTime=2
              Folder Alturas
                If barrenoActual≟1 or barrenoActual≟3 or barrenoActual≟5 or barrenoActual≟7 or barrenoActual≟9 or barrenoActual≟11 or barrenoActual≟13 or barrenoActual≟15 or barrenoActual≟17 or barrenoActual≟19 or barrenoActual≟21 or barrenoActual≟23 or barrenoActual≟25 or barrenoActual≟27
                  Set ExpressionOutput pin=mensaje_mw10; expression=200
                  Wait DigitalInput pin=Continuar_M30; digitalValue=1
                  Wait Sleep waitTime=1
                  Set ExpressionOutput pin=mensaje_mw10; expression=150
                  Wait Sleep waitTime=1
                MoveJ speed 30 deg/s, acceleration 40 deg/s^2 (useActiveTCP=true) feature=Base
                  Waypoint Waypoint (Variable): variable=internos
                Wait Sleep waitTime=2
                If P1h[2]<P2h[2]
                  acomodo := (altura/(barrenosTotales-1))*(barrenoActual-1)
                  tcp := get_actual_tcp_pose()
                  offset_altura := p[tcp[0],tcp[1],((alta-0.0095)-(acomodo/1000)),tcp[3],tcp[4],tcp[5]]
                  MoveL speed 250 mm/s, acceleration 1200 mm/s^2 (useActiveTCP=true) feature=Base
                    Waypoint Waypoint (Variable): motionParameters(jointSpeed=1.047198 jointAcceleration=1.396263 cartesianSpeed=0.03 cartesianAcceleration=0.04); variable=offset_altura
                Else 
                  acomodo := (altura/(barrenosTotales-1))*(26-(barrenoActual-1))
                  tcp := get_actual_tcp_pose()
                  offset_altura := p[tcp[0],tcp[1],((alta-0.0095)-(acomodo/1000)),tcp[3],tcp[4],tcp[5]]
                  MoveL speed 250 mm/s, acceleration 1200 mm/s^2 (useActiveTCP=true) feature=Base
                    Waypoint Waypoint (Variable): motionParameters(jointSpeed=1.047198 jointAcceleration=1.396263 cartesianSpeed=0.03 cartesianAcceleration=0.04); variable=offset_altura
              Folder Freemove
                Wait Sleep waitTime=2
                Script: freedrive_mode()
                Wait Sleep waitTime=2.5
                Script: end_freedrive_mode()
              Wait Sleep waitTime=0.3
              Set DigitalOutput pin=config_out[1]; digitalValue=1
              Wait Sleep waitTime=1
              Wait Sleep waitTime=0.3
              Wait Sleep waitTime=0.3
              Wait Sleep waitTime=0.3
              Loop Counting (count=1) loopVariable(name=Loop_67)
                Poses_taladrado := pose_sub(get_actual_tcp_pose(), bajada_broca)
                Waypoint Waypoint (Variable): motionParameters(jointSpeed=1.047198 jointAcceleration=1.396263 cartesianSpeed=0.001 cartesianAcceleration=0.005); variable=Poses_taladrado
                If bajada_broca≟p[0,0,0.018,0,0,0]
                  num_barreno := str_cat("Barreno: ",barrenoActual)
                  tcp_actual := get_actual_tcp_pose()
                  X_actual := str_cat("     X: ",tcp_actual[0])
                  Y_actual := str_cat("     Y: ",tcp_actual[1])
                  pos_barreno := str_cat(X_actual,Y_actual)
                  Script: textmsg(num_barreno,pos_barreno)
                Poses_taladrado := pose_add(get_actual_tcp_pose(), bajada_broca)
                Waypoint Waypoint (Variable): motionParameters(jointSpeed=1.047198 jointAcceleration=1.396263 cartesianSpeed=0.01 cartesianAcceleration=0.01); variable=Poses_taladrado
                bajada_broca := pose_add(bajada_broca, p[0,0,0.018,0,0,0])
              MoveDirectionNode (selectedDirection=ZPlus toolParams=0.01, 0.01)
                Until DISTANCE (allowActions=false deceleration=3 distanceNodeType=STOP) Distance=0.05; motionParameters(blendRadius=0)
              MoveJ speed 30 deg/s, acceleration 40 deg/s^2 (useActiveTCP=true) feature=Base
                Waypoint Waypoint (Variable): variable=internos
              Wait Sleep waitTime=0.3
              Set DigitalOutput pin=config_out[1]; digitalValue=0
              Wait Sleep waitTime=0.3
              If barrenoActual≟13 or barrenoActual≟27
                MoveDirectionNode (selectedDirection=ZPlus toolParams=0.04, 0.03)
                  Until DISTANCE (allowActions=false deceleration=3 distanceNodeType=STOP) Distance=0.03; motionParameters(blendRadius=0)
                MoveJ speed 30 deg/s, acceleration 40 deg/s^2 (useActiveTCP=true) feature=Base
                  Waypoint Zona_der1: TCP in base x=-721.714 y=-174.597 z=506.289 mm, rx=2.1128 ry=-2.325 rz=0 rad; joints [0.057, -90.231, 90.368, -0.664, 90.292, 0.009] deg
                  Waypoint Posicion_Cero: TCP in base x=0.641 y=-324.742 z=1651.532 mm, rx=-0.0042 ry=-0.0154 rz=-3.0499 rad; joints [-0.001, -90.003, -0.001, -90, 0, 0.002] deg
                Call Quitar_Broca_Chida
                If barrenoActual≟13
                  Call Poner_Broca
                ElseIf barrenoActual≟27
                  Call Poner_Broca
                MoveJ speed 30 deg/s, acceleration 40 deg/s^2 (useActiveTCP=true) feature=Base
                  Waypoint Posicion_Cero: TCP in base x=0.641 y=-324.742 z=1651.532 mm, rx=-0.0042 ry=-0.0154 rz=-3.0499 rad; joints [-0.001, -90.003, -0.001, -90, 0, 0.002] deg
                  Waypoint Zona_der1: TCP in base x=-721.714 y=-174.597 z=506.289 mm, rx=2.1128 ry=-2.325 rz=0 rad; joints [0.057, -90.231, 90.368, -0.664, 90.292, 0.009] deg
              barrenoActual := barrenoActual+1
        Folder Linea 2 a 217
          broca := 217
          Folder Buje_inicial
            Buje_Inicial := L2B2
          Folder Buje_final
            Buje_Final := L2B1
          barrenosTotales := 27
          barrenoActual := 1
          Loop While (checkContinuously=false) expression=barrenoActual≤barrenosTotales
            MoveL speed 250 mm/s, acceleration 1200 mm/s^2 (useActiveTCP=true) feature=Base
              bajada_broca := p[0,0,0.018,0,0,0]
              internos := interpolate_pose(Buje_Inicial, Buje_Final, ((barrenoActual)-1)/((barrenosTotales)-1))
              Folder Alturas
                If barrenoActual≟1 or barrenoActual≟3 or barrenoActual≟5 or barrenoActual≟7 or barrenoActual≟9 or barrenoActual≟11 or barrenoActual≟13 or barrenoActual≟15 or barrenoActual≟17 or barrenoActual≟19 or barrenoActual≟21 or barrenoActual≟23 or barrenoActual≟25 or barrenoActual≟27
                  Set ExpressionOutput pin=mensaje_mw10; expression=200
                  Wait DigitalInput pin=Continuar_M30; digitalValue=1
                  Wait Sleep waitTime=1
                  Set ExpressionOutput pin=mensaje_mw10; expression=150
                  Wait Sleep waitTime=1
                MoveJ speed 30 deg/s, acceleration 40 deg/s^2 (useActiveTCP=true) feature=Base
                  Waypoint Waypoint (Variable): variable=internos
                Wait Sleep waitTime=2
                If P1h[2]<P2h[2]
                  acomodo := (altura/(barrenosTotales-1))*(barrenoActual-1)
                  tcp := get_actual_tcp_pose()
                  offset_altura := p[tcp[0],tcp[1],((alta-0.0095)-(acomodo/1000)),tcp[3],tcp[4],tcp[5]]
                  MoveL speed 250 mm/s, acceleration 1200 mm/s^2 (useActiveTCP=true) feature=Base
                    Waypoint Waypoint (Variable): motionParameters(jointSpeed=1.047198 jointAcceleration=1.396263 cartesianSpeed=0.03 cartesianAcceleration=0.04); variable=offset_altura
                Else 
                  acomodo := (altura/(barrenosTotales-1))*(26-(barrenoActual-1))
                  tcp := get_actual_tcp_pose()
                  offset_altura := p[tcp[0],tcp[1],((alta-0.0095)-(acomodo/1000)),tcp[3],tcp[4],tcp[5]]
                  MoveL speed 250 mm/s, acceleration 1200 mm/s^2 (useActiveTCP=true) feature=Base
                    Waypoint Waypoint (Variable): motionParameters(jointSpeed=1.047198 jointAcceleration=1.396263 cartesianSpeed=0.03 cartesianAcceleration=0.04); variable=offset_altura
              Folder Freemove
                Wait Sleep waitTime=2
                Script: freedrive_mode()
                Wait Sleep waitTime=2.5
                Script: end_freedrive_mode()
              Wait Sleep waitTime=0.3
              Set DigitalOutput pin=config_out[1]; digitalValue=1
              Wait Sleep waitTime=1
              Wait Sleep waitTime=0.3
              Wait Sleep waitTime=0.3
              Wait Sleep waitTime=0.3
              Loop Counting (count=1) loopVariable(name=Loop_69)
                Poses_taladrado := pose_sub(get_actual_tcp_pose(), bajada_broca)
                Waypoint Waypoint (Variable): motionParameters(jointSpeed=1.047198 jointAcceleration=1.396263 cartesianSpeed=0.001 cartesianAcceleration=0.005); variable=Poses_taladrado
                If bajada_broca≟p[0,0,0.018,0,0,0]
                  num_barreno := str_cat("Barreno: ",barrenoActual)
                  tcp_actual := get_actual_tcp_pose()
                  X_actual := str_cat("     X: ",tcp_actual[0])
                  Y_actual := str_cat("     Y: ",tcp_actual[1])
                  pos_barreno := str_cat(X_actual,Y_actual)
                  Script: textmsg(num_barreno,pos_barreno)
                Poses_taladrado := pose_add(get_actual_tcp_pose(), bajada_broca)
                Waypoint Waypoint (Variable): motionParameters(jointSpeed=1.047198 jointAcceleration=1.396263 cartesianSpeed=0.01 cartesianAcceleration=0.01); variable=Poses_taladrado
                bajada_broca := pose_add(bajada_broca, p[0,0,0.018,0,0,0])
              MoveDirectionNode (selectedDirection=ZPlus toolParams=0.01, 0.01)
                Until DISTANCE (allowActions=false deceleration=3 distanceNodeType=STOP) Distance=0.05; motionParameters(blendRadius=0)
              MoveJ speed 30 deg/s, acceleration 40 deg/s^2 (useActiveTCP=true) feature=Base
                Waypoint Waypoint (Variable): variable=internos
              Wait Sleep waitTime=0.3
              Set DigitalOutput pin=config_out[1]; digitalValue=0
              Wait Sleep waitTime=0.3
              If barrenoActual≟13
                MoveDirectionNode (selectedDirection=ZPlus toolParams=0.03, 0.04)
                  Until DISTANCE (allowActions=false deceleration=3 distanceNodeType=STOP) Distance=0.03; motionParameters(blendRadius=0)
                MoveJ speed 60 deg/s, acceleration 80 deg/s^2 (useActiveTCP=true) feature=Base
                  Waypoint Zona_der1: TCP in base x=-721.714 y=-174.597 z=506.289 mm, rx=2.1128 ry=-2.325 rz=0 rad; joints [0.057, -90.231, 90.368, -0.664, 90.292, 0.009] deg
                  Waypoint Posicion_Cero: TCP in base x=0.641 y=-324.742 z=1651.532 mm, rx=-0.0042 ry=-0.0154 rz=-3.0499 rad; joints [-0.001, -90.003, -0.001, -90, 0, 0.002] deg
                Call Quitar_Broca_Chida
                Call Poner_Broca
                MoveJ speed 60 deg/s, acceleration 80 deg/s^2 (useActiveTCP=true) feature=Base
                  Waypoint Posicion_Cero: TCP in base x=0.641 y=-324.742 z=1651.532 mm, rx=-0.0042 ry=-0.0154 rz=-3.0499 rad; joints [-0.001, -90.003, -0.001, -90, 0, 0.002] deg
                  Waypoint Zona_der1: TCP in base x=-721.714 y=-174.597 z=506.289 mm, rx=2.1128 ry=-2.325 rz=0 rad; joints [0.057, -90.231, 90.368, -0.664, 90.292, 0.009] deg
              ElseIf barrenoActual≟27
                MoveDirectionNode (selectedDirection=ZPlus toolParams=0.03, 0.04)
                  Until DISTANCE (allowActions=false deceleration=3 distanceNodeType=STOP) Distance=0.03; motionParameters(blendRadius=0)
                MoveJ speed 60 deg/s, acceleration 80 deg/s^2 (useActiveTCP=true) feature=Base
                  Waypoint Zona_der1: TCP in base x=-721.714 y=-174.597 z=506.289 mm, rx=2.1128 ry=-2.325 rz=0 rad; joints [0.057, -90.231, 90.368, -0.664, 90.292, 0.009] deg
                  Waypoint Posicion_Cero: TCP in base x=0.641 y=-324.742 z=1651.532 mm, rx=-0.0042 ry=-0.0154 rz=-3.0499 rad; joints [-0.001, -90.003, -0.001, -90, 0, 0.002] deg
                Call Quitar_Broca_Chida
                Set DigitalOutput pin=carrusel_home; digitalValue=1
                Wait Sleep waitTime=1
                Set DigitalOutput pin=carrusel_home; digitalValue=0
                Set ExpressionOutput pin=mensaje_mw10; expression=120
                Wait DigitalInput pin=Continuar_M30; digitalValue=1
                Wait Sleep waitTime=1
                Set ExpressionOutput pin=mensaje_mw10; expression=100
                Wait DigitalInput pin=Continuar_M30; digitalValue=1
                Wait Sleep waitTime=1
                MoveJ speed 60 deg/s, acceleration 80 deg/s^2 (useActiveTCP=true) feature=Base
                  Waypoint Traslacion_der: TCP in base x=174.612 y=-721.747 z=506.267 mm, rx=3.1383 ry=-0.1432 rz=0.0001 rad; joints [89.991, -90.247, 90.386, -0.667, 89.974, 0.014] deg
              barrenoActual := barrenoActual+1
      Set DigitalOutput pin=pos1_term_m611; digitalValue=1
      Wait Sleep waitTime=1
      Set DigitalOutput pin=pos1_term_m611; digitalValue=0
    ElseIf pos_sig_der≟1
      Folder Arranque
        Set ExpressionOutput pin=mensaje_mw10; expression=15
        Wait DigitalInput pin=Continuar_M30; digitalValue=1
        Wait Sleep waitTime=1
        MoveJ speed 60 deg/s, acceleration 80 deg/s^2 (useActiveTCP=true) feature=Base
          Waypoint Off_derecha: TCP in base x=175.178 y=-46.666 z=17.814 mm, rx=-1.9982 ry=0.0913 rz=0.0579 rad; joints [90, -90, 154.891, 0, 90, 0.001] deg
        Set DigitalOutput pin=postrnas_m187; digitalValue=1
        Wait Sleep waitTime=1
        Set DigitalOutput pin=Home_M20; digitalValue=1
        Wait Sleep waitTime=1
        Set DigitalOutput pin=postrnas_m187; digitalValue=0
        Set DigitalOutput pin=Home_M20; digitalValue=0
        Set ExpressionOutput pin=mensaje_mw10; expression=20
        Wait DigitalInput pin=Continuar_M30; digitalValue=1
        Wait Sleep waitTime=1
      Folder Traslacion
        Set ExpressionOutput pin=mensaje_mw10; expression=25
        Wait DigitalInput pin=Continuar_M30; digitalValue=1
        Wait Sleep waitTime=1
        MoveJ speed 60 deg/s, acceleration 80 deg/s^2 (useActiveTCP=true) feature=Base
          Waypoint Waypoint_8: TCP in base x=175.237 y=-168.919 z=168.903 mm, rx=3.0585 ry=-0.1387 rz=0.0062 rad; joints [90.001, -160.001, 154.893, -0.003, 90, 0.003] deg
          Waypoint Traslacion_der: TCP in base x=174.612 y=-721.747 z=506.267 mm, rx=3.1383 ry=-0.1432 rz=0.0001 rad; joints [89.991, -90.247, 90.386, -0.667, 89.974, 0.014] deg
        Set ExpressionOutput pin=mensaje_mw10; expression=105
        Wait DigitalInput pin=Continuar_M30; digitalValue=1
        Wait Sleep waitTime=1
        Set ExpressionOutput pin=mensaje_mw10; expression=145
        Wait DigitalInput pin=Continuar_M30; digitalValue=1
        Wait Sleep waitTime=1
        Set DigitalOutput pin=postrnas_m187; digitalValue=1
        Wait Sleep waitTime=1
        Set DigitalOutput pin=pos2_der_mw698; digitalValue=1
        Wait Sleep waitTime=1
        Set DigitalOutput pin=pos2_der_mw698; digitalValue=0
        Set DigitalOutput pin=postrnas_m187; digitalValue=0
        Wait Sleep waitTime=10
      Folder Brocas
        Set DigitalOutput pin=carrusel_home; digitalValue=1
        Wait Sleep waitTime=1
        Set DigitalOutput pin=carrusel_home; digitalValue=0
        Set ExpressionOutput pin=mensaje_mw10; expression=40
        Wait DigitalInput pin=Continuar_M30; digitalValue=1
        Wait Sleep waitTime=1
        Set DigitalOutput pin=carrusel_home; digitalValue=1
        Wait Sleep waitTime=1
        Set DigitalOutput pin=carrusel_home; digitalValue=0
        Set ExpressionOutput pin=mensaje_mw10; expression=45
        Wait DigitalInput pin=Continuar_M30; digitalValue=1
        Wait Sleep waitTime=1
        Call Poner_Broca
      Folder Offsets factor
        SuppressedNode
          broca := 1645
        L1B1x := (((0.09525254)/(0.09525))*(0.09525254))*(1)
        L1B1y := (((-0.012)/(-0.0127))*(-0.012))*(1)
        L1B2x := (((0.74)/(0.75565))*(0.74))*(1.0003)
        L1B2y := (((-0.00986)/(-0.0127))*(-0.00986))*(1.0086956521739)
        L2B1x := ((0.09513062)/(0.09525))*(0.09525)
        L2B1y := ((0.39369238)/(0.3937))*(0.39369238)
        L2B2x := ((0.75565508)/(0.75565))*(0.75565508)
        L2B2y := ((0.39290032)/(0.3937))*(0.39290032)
      Folder Calibracion
        Set ExpressionOutput pin=mensaje_mw10; expression=50
        Wait DigitalInput pin=Continuar_M30; digitalValue=1
        Wait Sleep waitTime=1
        MoveJ speed 60 deg/s, acceleration 80 deg/s^2 (useActiveTCP=true) feature=Base
          Waypoint Posicion_Cero: TCP in base x=0.641 y=-324.742 z=1651.532 mm, rx=-0.0042 ry=-0.0154 rz=-3.0499 rad; joints [-0.001, -90.003, -0.001, -90, 0, 0.002] deg
          Waypoint Zona_der1: TCP in base x=-721.714 y=-174.597 z=506.289 mm, rx=2.1128 ry=-2.325 rz=0 rad; joints [0.057, -90.231, 90.368, -0.664, 90.292, 0.009] deg
        broca := 1645
        Set ExpressionOutput pin=mensaje_mw10; expression=125
        Wait DigitalInput pin=Continuar_M30; digitalValue=1
        Wait Sleep waitTime=1
        Set ExpressionOutput pin=mensaje_mw10; expression=130
        Wait DigitalInput pin=Continuar_M30; digitalValue=1
        Wait Sleep waitTime=1
        Call Calibracion
      Folder GoNoGo
        Set ExpressionOutput pin=mensaje_mw10; expression=55
        Wait DigitalInput pin=Continuar_M30; digitalValue=1
        Wait Sleep waitTime=1
        Set ExpressionOutput pin=mensaje_mw10; expression=60
        Wait DigitalInput pin=Continuar_M30; digitalValue=1
        Wait Sleep waitTime=1
        Folder Linea1_Buje1
          Xfin := (((L1B1x)*Xp)-(Xd)-((L1B1y)*(1/m2)))*(-1)
          Yfin := (((L1B1y)*Yp)-(Yd)+((L1B1x)*m1))*(-1)
          rotaciones := get_actual_tcp_pose()
          var_3 := rotaciones[3]
          var_4 := rotaciones[4]
          var_5 := rotaciones[5]
          If broca≟1645
            PosFinal := p[Xfin+0.00208915,Yfin+0.00208915,0.1,var_3,var_4,var_5]
          ElseIf broca≟1935
            PosFinal := p[Xfin+0.00245745,Yfin+0.00245745,0.1,var_3,var_4,var_5]
          ElseIf broca≟217
            PosFinal := p[Xfin+0.0027559,Yfin+0.0027559,0.1,var_3,var_4,var_5]
          Buje_Final := PosFinal
        MoveJ speed 60 deg/s, acceleration 80 deg/s^2 (useActiveTCP=true) feature=Base
          Waypoint Waypoint (Variable): variable=Buje_Final
        Wait Sleep waitTime=1
        Folder Alturas
          If P1h[2]<P2h[2]
            tcp := get_actual_tcp_pose()
            offset_altura := p[tcp[0],tcp[1],((alta-0.0095)-(altura/1000)),tcp[3],tcp[4],tcp[5]]
            MoveL speed 250 mm/s, acceleration 1200 mm/s^2 (useActiveTCP=true) feature=Base
              Waypoint Waypoint (Variable): motionParameters(jointSpeed=1.047198 jointAcceleration=1.396263 cartesianSpeed=0.03 cartesianAcceleration=0.04); variable=offset_altura
          Else 
            tcp := get_actual_tcp_pose()
            offset_altura := p[tcp[0],tcp[1],((alta-0.0095)),tcp[3],tcp[4],tcp[5]]
            MoveL speed 250 mm/s, acceleration 1200 mm/s^2 (useActiveTCP=true) feature=Base
              Waypoint Waypoint (Variable): motionParameters(jointSpeed=1.047198 jointAcceleration=1.396263 cartesianSpeed=0.03 cartesianAcceleration=0.04); variable=offset_altura
        MoveL speed 60 mm/s, acceleration 80 mm/s^2 (useActiveTCP=true) feature=Base
          Folder Freemove
            Wait Sleep waitTime=2
            Script: freedrive_mode()
            Wait Sleep waitTime=2.5
            Script: end_freedrive_mode()
            var_11 := get_actual_tcp_pose()
            var_11 := p[var_11[0]*1000,var_11[1]*1000,420,420,420,420]
            var_11 := get_actual_tcp_pose()
            var_11 := p[var_11[0],var_11[1],0.1,var_11[3],var_11[4],var_11[5]]
          MoveDirectionNode (selectedDirection=ZPlus)
            Until DISTANCE (allowActions=false deceleration=3 distanceNodeType=STOP) Distance=0.15; motionParameters(blendRadius=0)
          MoveDirectionNode (selectedDirection=XMinus)
            Until DISTANCE (allowActions=false deceleration=3 distanceNodeType=STOP) Distance=0.42; motionParameters(blendRadius=0)
        L1B1 := var_11
        Folder Linea1_Buje2
          Xfin := (((L1B2x)*Xp)-(Xd)-((L1B2y)*(1/m2)))*(-1)
          Yfin := (((L1B2y)*Yp)-(Yd)+((L1B2x)*m1))*(-1)
          rotaciones := get_actual_tcp_pose()
          var_3 := rotaciones[3]
          var_4 := rotaciones[4]
          var_5 := rotaciones[5]
          If broca≟1645
            PosFinal := p[Xfin+0.00208915,Yfin+0.00208915,0.1,var_3,var_4,var_5]
          ElseIf broca≟1935
            PosFinal := p[Xfin+0.00245745,Yfin+0.00245745,0.1,var_3,var_4,var_5]
          ElseIf broca≟217
            PosFinal := p[Xfin+0.0027559,Yfin+0.0027559,0.1,var_3,var_4,var_5]
          Buje_Final := PosFinal
        MoveJ speed 60 deg/s, acceleration 80 deg/s^2 (useActiveTCP=true) feature=Base
          Waypoint Waypoint (Variable): variable=Buje_Final
        Wait Sleep waitTime=1
        Folder Alturas
          If P1h[2]<P2h[2]
            tcp := get_actual_tcp_pose()
            offset_altura := p[tcp[0],tcp[1],((alta-0.0095)),tcp[3],tcp[4],tcp[5]]
            MoveL speed 250 mm/s, acceleration 1200 mm/s^2 (useActiveTCP=true) feature=Base
              Waypoint Waypoint (Variable): motionParameters(jointSpeed=1.047198 jointAcceleration=1.396263 cartesianSpeed=0.03 cartesianAcceleration=0.04); variable=offset_altura
          Else 
            tcp := get_actual_tcp_pose()
            offset_altura := p[tcp[0],tcp[1],((alta-0.0095)-(altura/1000)),tcp[3],tcp[4],tcp[5]]
            MoveL speed 250 mm/s, acceleration 1200 mm/s^2 (useActiveTCP=true) feature=Base
              Waypoint Waypoint (Variable): motionParameters(jointSpeed=1.047198 jointAcceleration=1.396263 cartesianSpeed=0.03 cartesianAcceleration=0.04); variable=offset_altura
        MoveL speed 60 mm/s, acceleration 80 mm/s^2 (useActiveTCP=true) feature=Base
          Folder Freemove
            Wait Sleep waitTime=2
            Script: freedrive_mode()
            Wait Sleep waitTime=2.5
            Script: end_freedrive_mode()
            var_11 := get_actual_tcp_pose()
            var_11 := p[var_11[0]*1000,var_11[1]*1000,420,420,420,420]
            var_11 := get_actual_tcp_pose()
            var_11 := p[var_11[0],var_11[1],0.1,var_11[3],var_11[4],var_11[5]]
          MoveDirectionNode (selectedDirection=ZPlus)
            Until DISTANCE (allowActions=false deceleration=3 distanceNodeType=STOP) Distance=0.15; motionParameters(blendRadius=0)
        L1B2 := var_11
        Folder Linea2_Buje2
          Xfin := (((L2B2x)*Xp)-(Xd)-((L2B2y)*(1/m2)))*(-1)
          Yfin := (((L2B2y)*Yp)-(Yd)+((L2B2x)*m1))*(-1)
          rotaciones := get_actual_tcp_pose()
          var_3 := rotaciones[3]
          var_4 := rotaciones[4]
          var_5 := rotaciones[5]
          If broca≟1645
            PosFinal := p[Xfin+0.00208915,Yfin+0.00208915,0.1,var_3,var_4,var_5]
          ElseIf broca≟1935
            PosFinal := p[Xfin+0.00245745,Yfin+0.00245745,0.1,var_3,var_4,var_5]
          ElseIf broca≟217
            PosFinal := p[Xfin+0.0027559,Yfin+0.0027559,0.1,var_3,var_4,var_5]
          Buje_Final := PosFinal
        MoveJ speed 60 deg/s, acceleration 80 deg/s^2 (useActiveTCP=true) feature=Base
          Waypoint Waypoint (Variable): variable=Buje_Final
        Wait Sleep waitTime=1
        Folder Alturas
          If P1h[2]<P2h[2]
            tcp := get_actual_tcp_pose()
            offset_altura := p[tcp[0],tcp[1],((alta-0.0095)),tcp[3],tcp[4],tcp[5]]
            MoveL speed 250 mm/s, acceleration 1200 mm/s^2 (useActiveTCP=true) feature=Base
              Waypoint Waypoint (Variable): motionParameters(jointSpeed=1.047198 jointAcceleration=1.396263 cartesianSpeed=0.03 cartesianAcceleration=0.04); variable=offset_altura
          Else 
            tcp := get_actual_tcp_pose()
            offset_altura := p[tcp[0],tcp[1],((alta-0.0095)-(altura/1000)),tcp[3],tcp[4],tcp[5]]
            MoveL speed 250 mm/s, acceleration 1200 mm/s^2 (useActiveTCP=true) feature=Base
              Waypoint Waypoint (Variable): motionParameters(jointSpeed=1.047198 jointAcceleration=1.396263 cartesianSpeed=0.03 cartesianAcceleration=0.04); variable=offset_altura
        MoveL speed 60 mm/s, acceleration 80 mm/s^2 (useActiveTCP=true) feature=Base
          Folder Freemove
            Wait Sleep waitTime=2
            Script: freedrive_mode()
            Wait Sleep waitTime=2.5
            Script: end_freedrive_mode()
            var_11 := get_actual_tcp_pose()
            var_11 := p[var_11[0]*1000,var_11[1]*1000,420,420,420,420]
            var_11 := get_actual_tcp_pose()
            var_11 := p[var_11[0],var_11[1],0.1,var_11[3],var_11[4],var_11[5]]
          MoveDirectionNode (selectedDirection=ZPlus)
            Until DISTANCE (allowActions=false deceleration=3 distanceNodeType=STOP) Distance=0.15; motionParameters(blendRadius=0)
        L2B2 := var_11
        Folder Linea2_Buje1
          Xfin := (((L2B1x)*Xp)-(Xd)-((L2B1y)*(1/m2)))*(-1)
          Yfin := (((L2B1y)*Yp)-(Yd)+((L2B1x)*m1))*(-1)
          rotaciones := get_actual_tcp_pose()
          var_3 := rotaciones[3]
          var_4 := rotaciones[4]
          var_5 := rotaciones[5]
          If broca≟1645
            PosFinal := p[Xfin+0.00208915,Yfin+0.00208915,0.1,var_3,var_4,var_5]
          ElseIf broca≟1935
            PosFinal := p[Xfin+0.00245745,Yfin+0.00245745,0.1,var_3,var_4,var_5]
          ElseIf broca≟217
            PosFinal := p[Xfin+0.0027559,Yfin+0.0027559,0.1,var_3,var_4,var_5]
          Buje_Final := PosFinal
        MoveJ speed 60 deg/s, acceleration 80 deg/s^2 (useActiveTCP=true) feature=Base
          Waypoint Waypoint (Variable): variable=Buje_Final
        Wait Sleep waitTime=1
        Folder Alturas
          If P1h[2]<P2h[2]
            tcp := get_actual_tcp_pose()
            offset_altura := p[tcp[0],tcp[1],((alta-0.0095)-(altura/1000)),tcp[3],tcp[4],tcp[5]]
            MoveL speed 250 mm/s, acceleration 1200 mm/s^2 (useActiveTCP=true) feature=Base
              Waypoint Waypoint (Variable): motionParameters(jointSpeed=1.047198 jointAcceleration=1.396263 cartesianSpeed=0.03 cartesianAcceleration=0.04); variable=offset_altura
          Else 
            tcp := get_actual_tcp_pose()
            offset_altura := p[tcp[0],tcp[1],((alta-0.0095)),tcp[3],tcp[4],tcp[5]]
            MoveL speed 250 mm/s, acceleration 1200 mm/s^2 (useActiveTCP=true) feature=Base
              Waypoint Waypoint (Variable): motionParameters(jointSpeed=1.047198 jointAcceleration=1.396263 cartesianSpeed=0.03 cartesianAcceleration=0.04); variable=offset_altura
        MoveL speed 60 mm/s, acceleration 80 mm/s^2 (useActiveTCP=true) feature=Base
          Folder Freemove
            Wait Sleep waitTime=2
            Script: freedrive_mode()
            Wait Sleep waitTime=2.5
            Script: end_freedrive_mode()
            var_11 := get_actual_tcp_pose()
            var_11 := p[var_11[0]*1000,var_11[1]*1000,420,420,420,420]
            var_11 := get_actual_tcp_pose()
            var_11 := p[var_11[0],var_11[1],0.1,var_11[3],var_11[4],var_11[5]]
          MoveDirectionNode (selectedDirection=ZPlus)
            Until DISTANCE (allowActions=false deceleration=3 distanceNodeType=STOP) Distance=0.15; motionParameters(blendRadius=0)
        L2B1 := var_11
        MoveJ speed 60 deg/s, acceleration 80 deg/s^2 (useActiveTCP=true) feature=Base
          Waypoint Zona_der1: TCP in base x=-721.714 y=-174.597 z=506.289 mm, rx=2.1128 ry=-2.325 rz=0 rad; joints [0.057, -90.231, 90.368, -0.664, 90.292, 0.009] deg
      SuppressedNode
        Folder Cancelar barrenacion
          MoveJ speed 60 deg/s, acceleration 80 deg/s^2 (useActiveTCP=true) feature=Base
            Waypoint Zona_der1: TCP in base x=-721.714 y=-174.597 z=506.289 mm, rx=2.1128 ry=-2.325 rz=0 rad; joints [0.057, -90.231, 90.368, -0.664, 90.292, 0.009] deg
            Waypoint Posicion_Cero: TCP in base x=0.641 y=-324.742 z=1651.532 mm, rx=-0.0042 ry=-0.0154 rz=-3.0499 rad; joints [-0.001, -90.003, -0.001, -90, 0, 0.002] deg
          Call Quitar_Broca_Chida
          Set DigitalOutput pin=lado_hecho; digitalValue=1
          Set ExpressionOutput pin=mensaje_mw10; expression=100
          Wait DigitalInput pin=Continuar_M30; digitalValue=1
          Wait Sleep waitTime=1
          Set ExpressionOutput pin=mensaje_mw10; expression=155
          Wait DigitalInput pin=Continuar_M30; digitalValue=1
          Wait Sleep waitTime=1
          Set ExpressionOutput pin=mensaje_mw10; expression=35
          Wait DigitalInput pin=Continuar_M30; digitalValue=1
          Wait Sleep waitTime=1
      Folder Colocar broca
        Call Quitar_Broca_Chida
        Call Poner_Broca
      Folder Barrenado
        Set ExpressionOutput pin=mensaje_mw10; expression=65
        Wait DigitalInput pin=Continuar_M30; digitalValue=1
        Wait Sleep waitTime=1
        Set ExpressionOutput pin=mensaje_mw10; expression=150
        Wait Sleep waitTime=1
        Folder Linea 1 a 1645
          broca := 1645
          Folder Buje_inicial
            Buje_Inicial := L1B2
          Folder Buje_final
            Buje_Final := L1B1
          barrenosTotales := 27
          barrenoActual := 1
          Loop While (checkContinuously=false) expression=barrenoActual≤barrenosTotales
            MoveL speed 250 mm/s, acceleration 1200 mm/s^2 (useActiveTCP=true) feature=Base
              bajada_broca := p[0,0,0.006,0,0,0]
              internos := interpolate_pose(Buje_Inicial, Buje_Final, ((barrenoActual)-1)/((barrenosTotales)-1))
              If barrenoActual≟1 or barrenoActual≟3 or barrenoActual≟5 or barrenoActual≟7 or barrenoActual≟9 or barrenoActual≟11 or barrenoActual≟13 or barrenoActual≟15 or barrenoActual≟17 or barrenoActual≟19 or barrenoActual≟21 or barrenoActual≟23 or barrenoActual≟25 or barrenoActual≟27
                Set ExpressionOutput pin=mensaje_mw10; expression=200
                Wait DigitalInput pin=Continuar_M30; digitalValue=1
                Wait Sleep waitTime=1
                Set ExpressionOutput pin=mensaje_mw10; expression=150
                Wait Sleep waitTime=1
              MoveJ speed 30 deg/s, acceleration 40 deg/s^2 (useActiveTCP=true) feature=Base
                Waypoint Waypoint (Variable): variable=internos
              Wait Sleep waitTime=2
              Folder Alturas
                If P1h[2]<P2h[2]
                  acomodo := (altura/(barrenosTotales-1))*(barrenoActual-1)
                  tcp := get_actual_tcp_pose()
                  offset_altura := p[tcp[0],tcp[1],((alta-0.0095)-(acomodo/1000)),tcp[3],tcp[4],tcp[5]]
                  MoveL speed 250 mm/s, acceleration 1200 mm/s^2 (useActiveTCP=true) feature=Base
                    Waypoint Waypoint (Variable): motionParameters(jointSpeed=1.047198 jointAcceleration=1.396263 cartesianSpeed=0.03 cartesianAcceleration=0.04); variable=offset_altura
                Else 
                  acomodo := (altura/(barrenosTotales-1))*(26-(barrenoActual-1))
                  tcp := get_actual_tcp_pose()
                  offset_altura := p[tcp[0],tcp[1],((alta-0.0095)-(acomodo/1000)),tcp[3],tcp[4],tcp[5]]
                  MoveL speed 250 mm/s, acceleration 1200 mm/s^2 (useActiveTCP=true) feature=Base
                    Waypoint Waypoint (Variable): motionParameters(jointSpeed=1.047198 jointAcceleration=1.396263 cartesianSpeed=0.03 cartesianAcceleration=0.04); variable=offset_altura
              Folder Freemove
                Wait Sleep waitTime=2
                Script: freedrive_mode()
                Wait Sleep waitTime=2.5
                Script: end_freedrive_mode()
              Wait Sleep waitTime=0.3
              Set DigitalOutput pin=config_out[1]; digitalValue=1
              Wait Sleep waitTime=1
              Wait Sleep waitTime=0.3
              Wait Sleep waitTime=0.3
              Wait Sleep waitTime=0.3
              Loop Counting (count=3) loopVariable(name=Loop_42)
                Poses_taladrado := pose_sub(get_actual_tcp_pose(), bajada_broca)
                Waypoint Waypoint (Variable): motionParameters(jointSpeed=1.047198 jointAcceleration=1.396263 cartesianSpeed=0.001 cartesianAcceleration=0.005); variable=Poses_taladrado
                If bajada_broca≟p[0,0,0.018,0,0,0]
                  num_barreno := str_cat("Barreno: ",barrenoActual)
                  tcp_actual := get_actual_tcp_pose()
                  X_actual := str_cat("     X: ",tcp_actual[0])
                  Y_actual := str_cat("     Y: ",tcp_actual[1])
                  pos_barreno := str_cat(X_actual,Y_actual)
                  Script: textmsg(num_barreno,pos_barreno)
                Poses_taladrado := pose_add(get_actual_tcp_pose(), bajada_broca)
                Waypoint Waypoint (Variable): motionParameters(jointSpeed=1.047198 jointAcceleration=1.396263 cartesianSpeed=0.01 cartesianAcceleration=0.01); variable=Poses_taladrado
                bajada_broca := pose_add(bajada_broca, p[0,0,0.006,0,0,0])
              MoveDirectionNode (selectedDirection=ZPlus toolParams=0.03, 0.04)
                Until DISTANCE (allowActions=false deceleration=3 distanceNodeType=STOP) Distance=0.05; motionParameters(blendRadius=0)
              MoveJ speed 30 deg/s, acceleration 40 deg/s^2 (useActiveTCP=true) feature=Base
                Waypoint Waypoint (Variable): variable=internos
              Wait Sleep waitTime=0.3
              Set DigitalOutput pin=config_out[1]; digitalValue=0
              Wait Sleep waitTime=0.3
              If barrenoActual≟13 or barrenoActual≟27
                MoveDirectionNode (selectedDirection=ZPlus toolParams=0.03, 0.04)
                  Until DISTANCE (allowActions=false deceleration=3 distanceNodeType=STOP) Distance=0.03; motionParameters(blendRadius=0)
                MoveJ speed 30 deg/s, acceleration 40 deg/s^2 (useActiveTCP=true) feature=Base
                  Waypoint Zona_der1: TCP in base x=-721.714 y=-174.597 z=506.289 mm, rx=2.1128 ry=-2.325 rz=0 rad; joints [0.057, -90.231, 90.368, -0.664, 90.292, 0.009] deg
                  Waypoint Posicion_Cero: TCP in base x=0.641 y=-324.742 z=1651.532 mm, rx=-0.0042 ry=-0.0154 rz=-3.0499 rad; joints [-0.001, -90.003, -0.001, -90, 0, 0.002] deg
                Call Quitar_Broca_Chida
                If barrenoActual≟13
                  Call Poner_Broca
                ElseIf barrenoActual≟27
                  Call Poner_Broca
                MoveJ speed 30 deg/s, acceleration 40 deg/s^2 (useActiveTCP=true) feature=Base
                  Waypoint Posicion_Cero: TCP in base x=0.641 y=-324.742 z=1651.532 mm, rx=-0.0042 ry=-0.0154 rz=-3.0499 rad; joints [-0.001, -90.003, -0.001, -90, 0, 0.002] deg
                  Waypoint Zona_der1: TCP in base x=-721.714 y=-174.597 z=506.289 mm, rx=2.1128 ry=-2.325 rz=0 rad; joints [0.057, -90.231, 90.368, -0.664, 90.292, 0.009] deg
              barrenoActual := barrenoActual+1
        Folder Linea 2 a 1645
          broca := 1645
          Folder Buje_inicial
            Buje_Inicial := L2B2
          Folder Buje_final
            Buje_Final := L2B1
          barrenosTotales := 27
          barrenoActual := 1
          Loop While (checkContinuously=false) expression=barrenoActual≤barrenosTotales
            MoveL speed 250 mm/s, acceleration 1200 mm/s^2 (useActiveTCP=true) feature=Base
              bajada_broca := p[0,0,0.006,0,0,0]
              internos := interpolate_pose(Buje_Inicial, Buje_Final, ((barrenoActual)-1)/((barrenosTotales)-1))
              Folder Alturas
                If barrenoActual≟1 or barrenoActual≟3 or barrenoActual≟5 or barrenoActual≟7 or barrenoActual≟9 or barrenoActual≟11 or barrenoActual≟13 or barrenoActual≟15 or barrenoActual≟17 or barrenoActual≟19 or barrenoActual≟21 or barrenoActual≟23 or barrenoActual≟25 or barrenoActual≟27
                  Set ExpressionOutput pin=mensaje_mw10; expression=200
                  Wait DigitalInput pin=Continuar_M30; digitalValue=1
                  Wait Sleep waitTime=1
                  Set ExpressionOutput pin=mensaje_mw10; expression=150
                  Wait Sleep waitTime=1
                MoveJ speed 30 deg/s, acceleration 40 deg/s^2 (useActiveTCP=true) feature=Base
                  Waypoint Waypoint (Variable): variable=internos
                Wait Sleep waitTime=2
                If P1h[2]<P2h[2]
                  acomodo := (altura/(barrenosTotales-1))*(barrenoActual-1)
                  tcp := get_actual_tcp_pose()
                  offset_altura := p[tcp[0],tcp[1],((alta-0.0095)-(acomodo/1000)),tcp[3],tcp[4],tcp[5]]
                  MoveL speed 250 mm/s, acceleration 1200 mm/s^2 (useActiveTCP=true) feature=Base
                    Waypoint Waypoint (Variable): motionParameters(jointSpeed=1.047198 jointAcceleration=1.396263 cartesianSpeed=0.03 cartesianAcceleration=0.04); variable=offset_altura
                Else 
                  acomodo := (altura/(barrenosTotales-1))*(26-(barrenoActual-1))
                  tcp := get_actual_tcp_pose()
                  offset_altura := p[tcp[0],tcp[1],((alta-0.0095)-(acomodo/1000)),tcp[3],tcp[4],tcp[5]]
                  MoveL speed 250 mm/s, acceleration 1200 mm/s^2 (useActiveTCP=true) feature=Base
                    Waypoint Waypoint (Variable): motionParameters(jointSpeed=1.047198 jointAcceleration=1.396263 cartesianSpeed=0.03 cartesianAcceleration=0.04); variable=offset_altura
              Folder Freemove
                Wait Sleep waitTime=2
                Script: freedrive_mode()
                Wait Sleep waitTime=2.5
                Script: end_freedrive_mode()
              Wait Sleep waitTime=0.3
              Set DigitalOutput pin=config_out[1]; digitalValue=1
              Wait Sleep waitTime=1
              Wait Sleep waitTime=0.3
              Wait Sleep waitTime=0.3
              Wait Sleep waitTime=0.3
              Loop Counting (count=3) loopVariable(name=Loop_46)
                Poses_taladrado := pose_sub(get_actual_tcp_pose(), bajada_broca)
                Waypoint Waypoint (Variable): motionParameters(jointSpeed=1.047198 jointAcceleration=1.396263 cartesianSpeed=0.001 cartesianAcceleration=0.005); variable=Poses_taladrado
                If bajada_broca≟p[0,0,0.018,0,0,0]
                  num_barreno := str_cat("Barreno: ",barrenoActual)
                  tcp_actual := get_actual_tcp_pose()
                  X_actual := str_cat("     X: ",tcp_actual[0])
                  Y_actual := str_cat("     Y: ",tcp_actual[1])
                  pos_barreno := str_cat(X_actual,Y_actual)
                  Script: textmsg(num_barreno,pos_barreno)
                Poses_taladrado := pose_add(get_actual_tcp_pose(), bajada_broca)
                Waypoint Waypoint (Variable): motionParameters(jointSpeed=1.047198 jointAcceleration=1.396263 cartesianSpeed=0.01 cartesianAcceleration=0.01); variable=Poses_taladrado
                bajada_broca := pose_add(bajada_broca, p[0,0,0.006,0,0,0])
              MoveDirectionNode (selectedDirection=ZPlus toolParams=0.03, 0.04)
                Until DISTANCE (allowActions=false deceleration=3 distanceNodeType=STOP) Distance=0.05; motionParameters(blendRadius=0)
              MoveJ speed 30 deg/s, acceleration 40 deg/s^2 (useActiveTCP=true) feature=Base
                Waypoint Waypoint (Variable): variable=internos
              Wait Sleep waitTime=0.3
              Set DigitalOutput pin=config_out[1]; digitalValue=0
              Wait Sleep waitTime=0.3
              If barrenoActual≟13
                MoveDirectionNode (selectedDirection=ZPlus)
                  Until DISTANCE (allowActions=false deceleration=3 distanceNodeType=STOP) Distance=0.03; motionParameters(blendRadius=0)
                MoveJ speed 60 deg/s, acceleration 80 deg/s^2 (useActiveTCP=true) feature=Base
                  Waypoint Zona_der1: TCP in base x=-721.714 y=-174.597 z=506.289 mm, rx=2.1128 ry=-2.325 rz=0 rad; joints [0.057, -90.231, 90.368, -0.664, 90.292, 0.009] deg
                  Waypoint Posicion_Cero: TCP in base x=0.641 y=-324.742 z=1651.532 mm, rx=-0.0042 ry=-0.0154 rz=-3.0499 rad; joints [-0.001, -90.003, -0.001, -90, 0, 0.002] deg
                Call Quitar_Broca_Chida
                Call Poner_Broca
                MoveJ speed 60 deg/s, acceleration 80 deg/s^2 (useActiveTCP=true) feature=Base
                  Waypoint Posicion_Cero: TCP in base x=0.641 y=-324.742 z=1651.532 mm, rx=-0.0042 ry=-0.0154 rz=-3.0499 rad; joints [-0.001, -90.003, -0.001, -90, 0, 0.002] deg
                  Waypoint Zona_der1: TCP in base x=-721.714 y=-174.597 z=506.289 mm, rx=2.1128 ry=-2.325 rz=0 rad; joints [0.057, -90.231, 90.368, -0.664, 90.292, 0.009] deg
              ElseIf barrenoActual≟27
                MoveDirectionNode (selectedDirection=ZPlus)
                  Until DISTANCE (allowActions=false deceleration=3 distanceNodeType=STOP) Distance=0.03; motionParameters(blendRadius=0)
                MoveJ speed 60 deg/s, acceleration 80 deg/s^2 (useActiveTCP=true) feature=Base
                  Waypoint Zona_der1: TCP in base x=-721.714 y=-174.597 z=506.289 mm, rx=2.1128 ry=-2.325 rz=0 rad; joints [0.057, -90.231, 90.368, -0.664, 90.292, 0.009] deg
                  Waypoint Posicion_Cero: TCP in base x=0.641 y=-324.742 z=1651.532 mm, rx=-0.0042 ry=-0.0154 rz=-3.0499 rad; joints [-0.001, -90.003, -0.001, -90, 0, 0.002] deg
                Call Quitar_Broca_Chida
                Set DigitalOutput pin=carrusel_home; digitalValue=1
                Wait Sleep waitTime=1
                Set DigitalOutput pin=carrusel_home; digitalValue=0
                Set ExpressionOutput pin=mensaje_mw10; expression=70
                Wait DigitalInput pin=Continuar_M30; digitalValue=1
                Wait Sleep waitTime=1
                Set ExpressionOutput pin=mensaje_mw10; expression=120
                Wait DigitalInput pin=Continuar_M30; digitalValue=1
                Wait Sleep waitTime=1
                Set DigitalOutput pin=carrusel_home; digitalValue=1
                Wait Sleep waitTime=1
                Set DigitalOutput pin=carrusel_home; digitalValue=0
                Set ExpressionOutput pin=mensaje_mw10; expression=75
                Wait DigitalInput pin=Continuar_M30; digitalValue=1
                Wait Sleep waitTime=1
                Call Poner_Broca
                broca := 1935
                MoveJ speed 60 deg/s, acceleration 80 deg/s^2 (useActiveTCP=true) feature=Base
                  Waypoint Posicion_Cero: TCP in base x=0.641 y=-324.742 z=1651.532 mm, rx=-0.0042 ry=-0.0154 rz=-3.0499 rad; joints [-0.001, -90.003, -0.001, -90, 0, 0.002] deg
                  Waypoint Zona_der1: TCP in base x=-721.714 y=-174.597 z=506.289 mm, rx=2.1128 ry=-2.325 rz=0 rad; joints [0.057, -90.231, 90.368, -0.664, 90.292, 0.009] deg
                Set ExpressionOutput pin=mensaje_mw10; expression=80
                Wait DigitalInput pin=Continuar_M30; digitalValue=1
                Wait Sleep waitTime=1
                Set ExpressionOutput pin=mensaje_mw10; expression=150
                Wait DigitalInput pin=Continuar_M30; digitalValue=1
                Wait Sleep waitTime=1
              barrenoActual := barrenoActual+1
        Folder Linea 1 a 1935
          broca := 1935
          Folder Buje_inicial
            Buje_Inicial := L1B2
          Folder Buje_final
            Buje_Final := L1B1
          barrenosTotales := 27
          barrenoActual := 1
          Loop While (checkContinuously=false) expression=barrenoActual≤barrenosTotales
            MoveL speed 250 mm/s, acceleration 1200 mm/s^2 (useActiveTCP=true) feature=Base
              bajada_broca := p[0,0,0.009,0,0,0]
              internos := interpolate_pose(Buje_Inicial, Buje_Final, ((barrenoActual)-1)/((barrenosTotales)-1))
              Folder Alturas
                If barrenoActual≟1 or barrenoActual≟3 or barrenoActual≟5 or barrenoActual≟7 or barrenoActual≟9 or barrenoActual≟11 or barrenoActual≟13 or barrenoActual≟15 or barrenoActual≟17 or barrenoActual≟19 or barrenoActual≟21 or barrenoActual≟23 or barrenoActual≟25 or barrenoActual≟27
                  Set ExpressionOutput pin=mensaje_mw10; expression=200
                  Wait DigitalInput pin=Continuar_M30; digitalValue=1
                  Wait Sleep waitTime=1
                  Set ExpressionOutput pin=mensaje_mw10; expression=150
                  Wait Sleep waitTime=1
                MoveJ speed 30 deg/s, acceleration 40 deg/s^2 (useActiveTCP=true) feature=Base
                  Waypoint Waypoint (Variable): variable=internos
                Wait Sleep waitTime=2
                If P1h[2]<P2h[2]
                  acomodo := (altura/(barrenosTotales-1))*(barrenoActual-1)
                  tcp := get_actual_tcp_pose()
                  offset_altura := p[tcp[0],tcp[1],((alta-0.0095)-(acomodo/1000)),tcp[3],tcp[4],tcp[5]]
                  MoveL speed 250 mm/s, acceleration 1200 mm/s^2 (useActiveTCP=true) feature=Base
                    Waypoint Waypoint (Variable): motionParameters(jointSpeed=1.047198 jointAcceleration=1.396263 cartesianSpeed=0.03 cartesianAcceleration=0.04); variable=offset_altura
                Else 
                  acomodo := (altura/(barrenosTotales-1))*(26-(barrenoActual-1))
                  tcp := get_actual_tcp_pose()
                  offset_altura := p[tcp[0],tcp[1],((alta-0.0095)-(acomodo/1000)),tcp[3],tcp[4],tcp[5]]
                  MoveL speed 250 mm/s, acceleration 1200 mm/s^2 (useActiveTCP=true) feature=Base
                    Waypoint Waypoint (Variable): motionParameters(jointSpeed=1.047198 jointAcceleration=1.396263 cartesianSpeed=0.03 cartesianAcceleration=0.04); variable=offset_altura
              Folder Freemove
                Wait Sleep waitTime=2
                Script: freedrive_mode()
                Wait Sleep waitTime=2.5
                Script: end_freedrive_mode()
              Wait Sleep waitTime=0.3
              Set DigitalOutput pin=config_out[1]; digitalValue=1
              Wait Sleep waitTime=1
              Wait Sleep waitTime=0.3
              Wait Sleep waitTime=0.3
              Wait Sleep waitTime=0.3
              Loop Counting (count=2) loopVariable(name=Loop_50)
                Poses_taladrado := pose_sub(get_actual_tcp_pose(), bajada_broca)
                Waypoint Waypoint (Variable): motionParameters(jointSpeed=1.047198 jointAcceleration=1.396263 cartesianSpeed=0.001 cartesianAcceleration=0.005); variable=Poses_taladrado
                If bajada_broca≟p[0,0,0.018,0,0,0]
                  num_barreno := str_cat("Barreno: ",barrenoActual)
                  tcp_actual := get_actual_tcp_pose()
                  X_actual := str_cat("     X: ",tcp_actual[0])
                  Y_actual := str_cat("     Y: ",tcp_actual[1])
                  pos_barreno := str_cat(X_actual,Y_actual)
                  Script: textmsg(num_barreno,pos_barreno)
                Poses_taladrado := pose_add(get_actual_tcp_pose(), bajada_broca)
                Waypoint Waypoint (Variable): motionParameters(jointSpeed=1.047198 jointAcceleration=1.396263 cartesianSpeed=0.01 cartesianAcceleration=0.01); variable=Poses_taladrado
                bajada_broca := pose_add(bajada_broca, p[0,0,0.009,0,0,0])
              MoveDirectionNode (selectedDirection=ZPlus toolParams=0.01, 0.01)
                Until DISTANCE (allowActions=false deceleration=3 distanceNodeType=STOP) Distance=0.05; motionParameters(blendRadius=0)
              MoveJ speed 30 deg/s, acceleration 40 deg/s^2 (useActiveTCP=true) feature=Base
                Waypoint Waypoint (Variable): variable=internos
              Wait Sleep waitTime=0.3
              Set DigitalOutput pin=config_out[1]; digitalValue=0
              Wait Sleep waitTime=0.3
              If barrenoActual≟13 or barrenoActual≟27
                MoveDirectionNode (selectedDirection=ZPlus toolParams=0.03, 0.04)
                  Until DISTANCE (allowActions=false deceleration=3 distanceNodeType=STOP) Distance=0.03; motionParameters(blendRadius=0)
                MoveJ speed 30 deg/s, acceleration 40 deg/s^2 (useActiveTCP=true) feature=Base
                  Waypoint Zona_der1: TCP in base x=-721.714 y=-174.597 z=506.289 mm, rx=2.1128 ry=-2.325 rz=0 rad; joints [0.057, -90.231, 90.368, -0.664, 90.292, 0.009] deg
                  Waypoint Posicion_Cero: TCP in base x=0.641 y=-324.742 z=1651.532 mm, rx=-0.0042 ry=-0.0154 rz=-3.0499 rad; joints [-0.001, -90.003, -0.001, -90, 0, 0.002] deg
                Call Quitar_Broca_Chida
                If barrenoActual≟13
                  Call Poner_Broca
                ElseIf barrenoActual≟27
                  Call Poner_Broca
                MoveJ speed 30 deg/s, acceleration 40 deg/s^2 (useActiveTCP=true) feature=Base
                  Waypoint Posicion_Cero: TCP in base x=0.641 y=-324.742 z=1651.532 mm, rx=-0.0042 ry=-0.0154 rz=-3.0499 rad; joints [-0.001, -90.003, -0.001, -90, 0, 0.002] deg
                  Waypoint Zona_der1: TCP in base x=-721.714 y=-174.597 z=506.289 mm, rx=2.1128 ry=-2.325 rz=0 rad; joints [0.057, -90.231, 90.368, -0.664, 90.292, 0.009] deg
              barrenoActual := barrenoActual+1
        Folder Linea 2 a 1935
          broca := 1935
          Folder Buje_inicial
            Buje_Inicial := L2B2
          Folder Buje_final
            Buje_Final := L2B1
          barrenosTotales := 27
          barrenoActual := 1
          Loop While (checkContinuously=false) expression=barrenoActual≤barrenosTotales
            MoveL speed 250 mm/s, acceleration 1200 mm/s^2 (useActiveTCP=true) feature=Base
              bajada_broca := p[0,0,0.009,0,0,0]
              internos := interpolate_pose(Buje_Inicial, Buje_Final, ((barrenoActual)-1)/((barrenosTotales)-1))
              Folder Alturas
                If barrenoActual≟1 or barrenoActual≟3 or barrenoActual≟5 or barrenoActual≟7 or barrenoActual≟9 or barrenoActual≟11 or barrenoActual≟13 or barrenoActual≟15 or barrenoActual≟17 or barrenoActual≟19 or barrenoActual≟21 or barrenoActual≟23 or barrenoActual≟25 or barrenoActual≟27
                  Set ExpressionOutput pin=mensaje_mw10; expression=200
                  Wait DigitalInput pin=Continuar_M30; digitalValue=1
                  Wait Sleep waitTime=1
                  Set ExpressionOutput pin=mensaje_mw10; expression=150
                  Wait Sleep waitTime=1
                MoveJ speed 30 deg/s, acceleration 40 deg/s^2 (useActiveTCP=true) feature=Base
                  Waypoint Waypoint (Variable): variable=internos
                Wait Sleep waitTime=2
                If P1h[2]<P2h[2]
                  acomodo := (altura/(barrenosTotales-1))*(barrenoActual-1)
                  tcp := get_actual_tcp_pose()
                  offset_altura := p[tcp[0],tcp[1],((alta-0.0095)-(acomodo/1000)),tcp[3],tcp[4],tcp[5]]
                  MoveL speed 250 mm/s, acceleration 1200 mm/s^2 (useActiveTCP=true) feature=Base
                    Waypoint Waypoint (Variable): motionParameters(jointSpeed=1.047198 jointAcceleration=1.396263 cartesianSpeed=0.03 cartesianAcceleration=0.04); variable=offset_altura
                Else 
                  acomodo := (altura/(barrenosTotales-1))*(26-(barrenoActual-1))
                  tcp := get_actual_tcp_pose()
                  offset_altura := p[tcp[0],tcp[1],((alta-0.0095)-(acomodo/1000)),tcp[3],tcp[4],tcp[5]]
                  MoveL speed 250 mm/s, acceleration 1200 mm/s^2 (useActiveTCP=true) feature=Base
                    Waypoint Waypoint (Variable): motionParameters(jointSpeed=1.047198 jointAcceleration=1.396263 cartesianSpeed=0.03 cartesianAcceleration=0.04); variable=offset_altura
              Folder Freemove
                Wait Sleep waitTime=2
                Script: freedrive_mode()
                Wait Sleep waitTime=2.5
                Script: end_freedrive_mode()
              Wait Sleep waitTime=0.3
              Set DigitalOutput pin=config_out[1]; digitalValue=1
              Wait Sleep waitTime=1
              Wait Sleep waitTime=0.3
              Wait Sleep waitTime=0.3
              Wait Sleep waitTime=0.3
              Loop Counting (count=2) loopVariable(name=Loop_54)
                Poses_taladrado := pose_sub(get_actual_tcp_pose(), bajada_broca)
                Waypoint Waypoint (Variable): motionParameters(jointSpeed=1.047198 jointAcceleration=1.396263 cartesianSpeed=0.001 cartesianAcceleration=0.005); variable=Poses_taladrado
                If bajada_broca≟p[0,0,0.018,0,0,0]
                  num_barreno := str_cat("Barreno: ",barrenoActual)
                  tcp_actual := get_actual_tcp_pose()
                  X_actual := str_cat("     X: ",tcp_actual[0])
                  Y_actual := str_cat("     Y: ",tcp_actual[1])
                  pos_barreno := str_cat(X_actual,Y_actual)
                  Script: textmsg(num_barreno,pos_barreno)
                Poses_taladrado := pose_add(get_actual_tcp_pose(), bajada_broca)
                Waypoint Waypoint (Variable): motionParameters(jointSpeed=1.047198 jointAcceleration=1.396263 cartesianSpeed=0.01 cartesianAcceleration=0.01); variable=Poses_taladrado
                bajada_broca := pose_add(bajada_broca, p[0,0,0.009,0,0,0])
              MoveDirectionNode (selectedDirection=ZPlus toolParams=0.01, 0.01)
                Until DISTANCE (allowActions=false deceleration=3 distanceNodeType=STOP) Distance=0.05; motionParameters(blendRadius=0)
              MoveJ speed 30 deg/s, acceleration 40 deg/s^2 (useActiveTCP=true) feature=Base
                Waypoint Waypoint (Variable): variable=internos
              Wait Sleep waitTime=0.3
              Set DigitalOutput pin=config_out[1]; digitalValue=0
